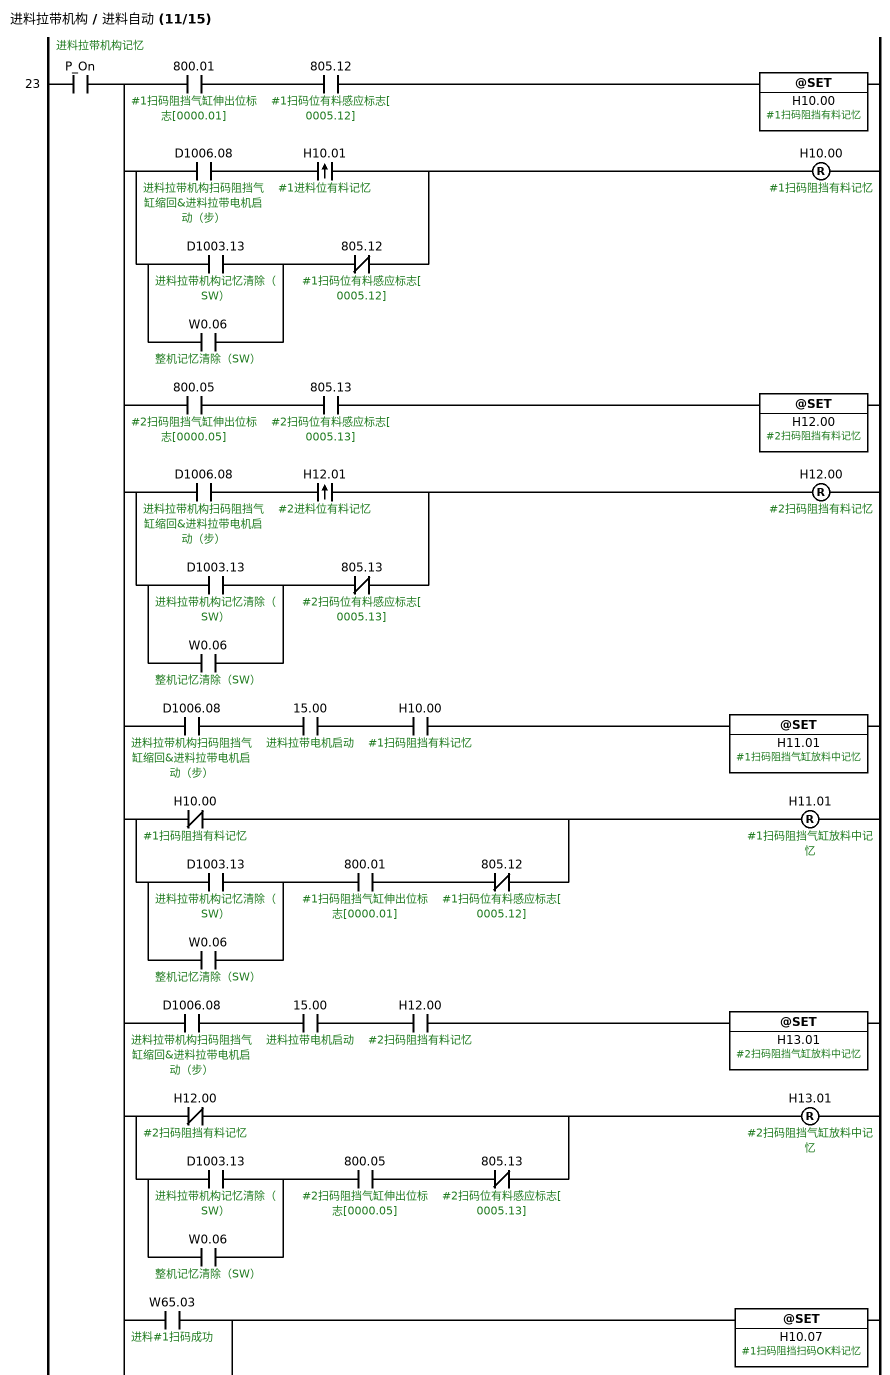
; [picture p48: 进料拉带机构 / 进料自动, rungs 23-23]

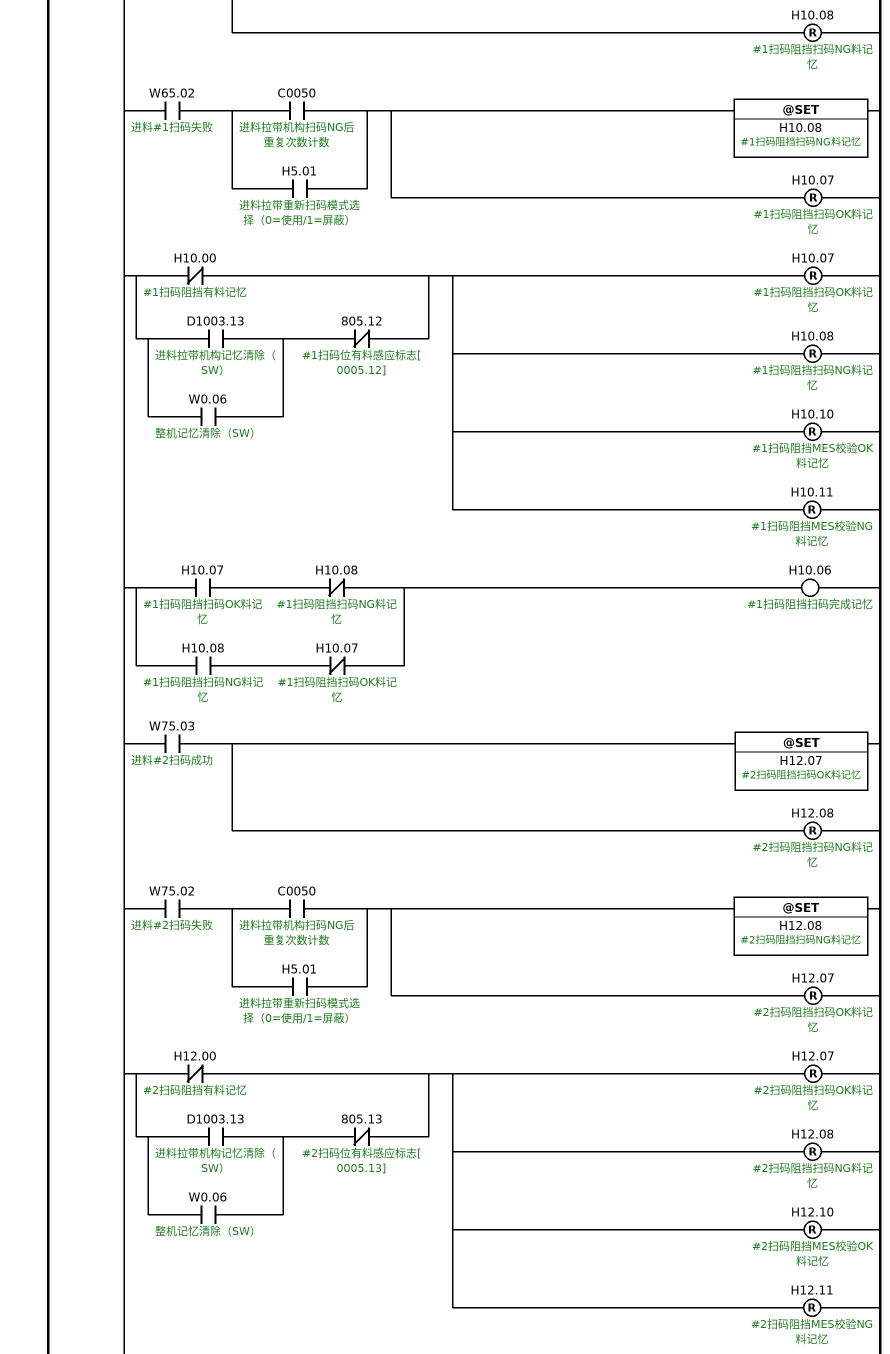

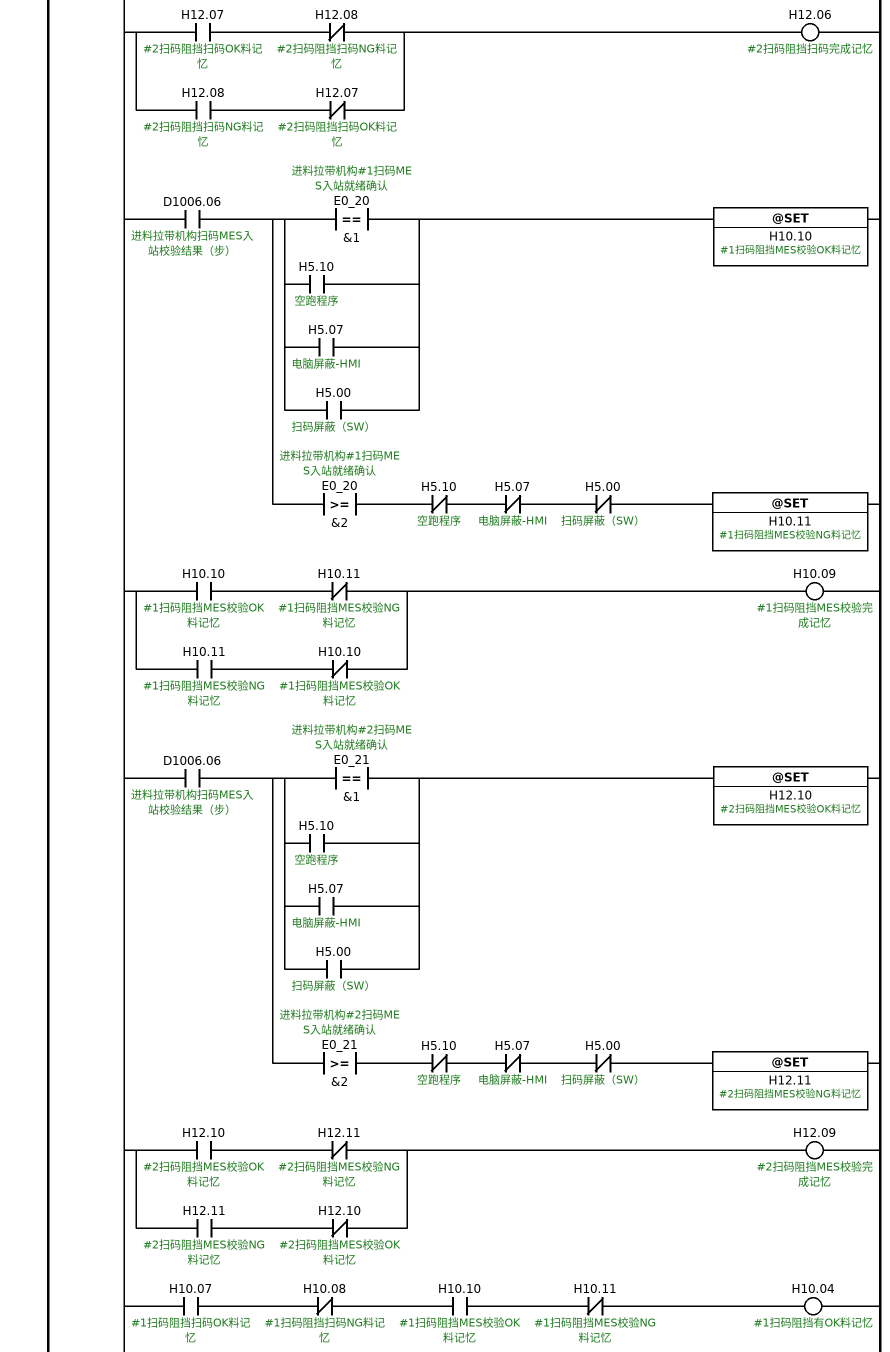

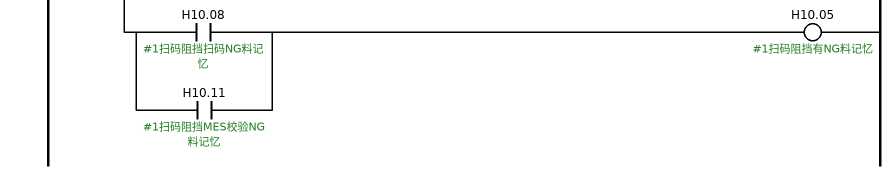
; rung 23: 进料拉带机构记忆
LD P_On
OUT TR0
AND 800.01  ; #1扫码阻挡气缸伸出位标志[0000.01]
AND 805.12  ; #1扫码位有料感应标志[0005.12]
@SET H10.00  ; #1扫码阻挡有料记忆
LD TR0
LD D1006.08  ; 进料拉带机构扫码阻挡气缸缩回&进料拉带电机启动（步）
@AND H10.01  ; #1进料位有料记忆
LD D1003.13  ; 进料拉带机构记忆清除（SW）
OR W0.06  ; 整机记忆清除（SW）
ANDNOT 805.12  ; #1扫码位有料感应标志[0005.12]
ORLD
ANDLD
RSET H10.00  ; #1扫码阻挡有料记忆
LD TR0
AND 800.05  ; #2扫码阻挡气缸伸出位标志[0000.05]
AND 805.13  ; #2扫码位有料感应标志[0005.13]
@SET H12.00  ; #2扫码阻挡有料记忆
LD TR0
LD D1006.08  ; 进料拉带机构扫码阻挡气缸缩回&进料拉带电机启动（步）
@AND H12.01  ; #2进料位有料记忆
LD D1003.13  ; 进料拉带机构记忆清除（SW）
OR W0.06  ; 整机记忆清除（SW）
ANDNOT 805.13  ; #2扫码位有料感应标志[0005.13]
ORLD
ANDLD
RSET H12.00  ; #2扫码阻挡有料记忆
LD TR0
AND D1006.08  ; 进料拉带机构扫码阻挡气缸缩回&进料拉带电机启动（步）
AND 15.00  ; 进料拉带电机启动
AND H10.00  ; #1扫码阻挡有料记忆
@SET H11.01  ; #1扫码阻挡气缸放料中记忆
LD TR0
LDNOT H10.00  ; #1扫码阻挡有料记忆
LD D1003.13  ; 进料拉带机构记忆清除（SW）
OR W0.06  ; 整机记忆清除（SW）
AND 800.01  ; #1扫码阻挡气缸伸出位标志[0000.01]
ANDNOT 805.12  ; #1扫码位有料感应标志[0005.12]
ORLD
ANDLD
RSET H11.01  ; #1扫码阻挡气缸放料中记忆
LD TR0
AND D1006.08  ; 进料拉带机构扫码阻挡气缸缩回&进料拉带电机启动（步）
AND 15.00  ; 进料拉带电机启动
AND H12.00  ; #2扫码阻挡有料记忆
@SET H13.01  ; #2扫码阻挡气缸放料中记忆
LD TR0
LDNOT H12.00  ; #2扫码阻挡有料记忆
LD D1003.13  ; 进料拉带机构记忆清除（SW）
OR W0.06  ; 整机记忆清除（SW）
AND 800.05  ; #2扫码阻挡气缸伸出位标志[0000.05]
ANDNOT 805.13  ; #2扫码位有料感应标志[0005.13]
ORLD
ANDLD
RSET H13.01  ; #2扫码阻挡气缸放料中记忆
LD TR0
AND W65.03  ; 进料#1扫码成功
@SET H10.07  ; #1扫码阻挡扫码OK料记忆
RSET H10.08  ; #1扫码阻挡扫码NG料记忆
LD TR0
AND W65.02  ; 进料#1扫码失败
LD C0050  ; 进料拉带机构扫码NG后重复次数计数
OR H5.01  ; 进料拉带重新扫码模式选择（0=使用/1=屏蔽）
ANDLD
@SET H10.08  ; #1扫码阻挡扫码NG料记忆
RSET H10.07  ; #1扫码阻挡扫码OK料记忆
LD TR0
LDNOT H10.00  ; #1扫码阻挡有料记忆
LD D1003.13  ; 进料拉带机构记忆清除（SW）
OR W0.06  ; 整机记忆清除（SW）
ANDNOT 805.12  ; #1扫码位有料感应标志[0005.12]
ORLD
ANDLD
RSET H10.07  ; #1扫码阻挡扫码OK料记忆
RSET H10.08  ; #1扫码阻挡扫码NG料记忆
RSET H10.10  ; #1扫码阻挡MES校验OK料记忆
RSET H10.11  ; #1扫码阻挡MES校验NG料记忆
LD TR0
LD H10.07  ; #1扫码阻挡扫码OK料记忆
ANDNOT H10.08  ; #1扫码阻挡扫码NG料记忆
LD H10.08  ; #1扫码阻挡扫码NG料记忆
ANDNOT H10.07  ; #1扫码阻挡扫码OK料记忆
ORLD
ANDLD
OUT H10.06  ; #1扫码阻挡扫码完成记忆
LD TR0
AND W75.03  ; 进料#2扫码成功
@SET H12.07  ; #2扫码阻挡扫码OK料记忆
RSET H12.08  ; #2扫码阻挡扫码NG料记忆
LD TR0
AND W75.02  ; 进料#2扫码失败
LD C0050  ; 进料拉带机构扫码NG后重复次数计数
OR H5.01  ; 进料拉带重新扫码模式选择（0=使用/1=屏蔽）
ANDLD
@SET H12.08  ; #2扫码阻挡扫码NG料记忆
RSET H12.07  ; #2扫码阻挡扫码OK料记忆
LD TR0
LDNOT H12.00  ; #2扫码阻挡有料记忆
LD D1003.13  ; 进料拉带机构记忆清除（SW）
OR W0.06  ; 整机记忆清除（SW）
ANDNOT 805.13  ; #2扫码位有料感应标志[0005.13]
ORLD
ANDLD
RSET H12.07  ; #2扫码阻挡扫码OK料记忆
RSET H12.08  ; #2扫码阻挡扫码NG料记忆
RSET H12.10  ; #2扫码阻挡MES校验OK料记忆
RSET H12.11  ; #2扫码阻挡MES校验NG料记忆
LD TR0
LD H12.07  ; #2扫码阻挡扫码OK料记忆
ANDNOT H12.08  ; #2扫码阻挡扫码NG料记忆
LD H12.08  ; #2扫码阻挡扫码NG料记忆
ANDNOT H12.07  ; #2扫码阻挡扫码OK料记忆
ORLD
ANDLD
OUT H12.06  ; #2扫码阻挡扫码完成记忆
LD TR0
AND D1006.06  ; 进料拉带机构扫码MES入站校验结果（步）
OUT TR1
LD=(300) E0_20 &1  ; 进料拉带机构#1扫码MES入站就绪确认  // 入站就绪确认=0：未确认，1：确认OK，2：确认NG
OR H5.10  ; 空跑程序
OR H5.07  ; 电脑屏蔽-HMI
OR H5.00  ; 扫码屏蔽（SW）
ANDLD
@SET H10.10  ; #1扫码阻挡MES校验OK料记忆
LD TR1
AND>=(325) E0_20 &2  ; 进料拉带机构#1扫码MES入站就绪确认  // 入站就绪确认=0：未确认，1：确认OK，2：确认NG
ANDNOT H5.10  ; 空跑程序
ANDNOT H5.07  ; 电脑屏蔽-HMI
ANDNOT H5.00  ; 扫码屏蔽（SW）
@SET H10.11  ; #1扫码阻挡MES校验NG料记忆
LD TR0
LD H10.10  ; #1扫码阻挡MES校验OK料记忆
ANDNOT H10.11  ; #1扫码阻挡MES校验NG料记忆
LD H10.11  ; #1扫码阻挡MES校验NG料记忆
ANDNOT H10.10  ; #1扫码阻挡MES校验OK料记忆
ORLD
ANDLD
OUT H10.09  ; #1扫码阻挡MES校验完成记忆
LD TR0
AND D1006.06  ; 进料拉带机构扫码MES入站校验结果（步）
OUT TR1
LD=(300) E0_21 &1  ; 进料拉带机构#2扫码MES入站就绪确认  // 入站就绪确认=0：未确认，1：确认OK，2：确认NG
OR H5.10  ; 空跑程序
OR H5.07  ; 电脑屏蔽-HMI
OR H5.00  ; 扫码屏蔽（SW）
ANDLD
@SET H12.10  ; #2扫码阻挡MES校验OK料记忆
LD TR1
AND>=(325) E0_21 &2  ; 进料拉带机构#2扫码MES入站就绪确认  // 入站就绪确认=0：未确认，1：确认OK，2：确认NG
ANDNOT H5.10  ; 空跑程序
ANDNOT H5.07  ; 电脑屏蔽-HMI
ANDNOT H5.00  ; 扫码屏蔽（SW）
@SET H12.11  ; #2扫码阻挡MES校验NG料记忆
LD TR0
LD H12.10  ; #2扫码阻挡MES校验OK料记忆
ANDNOT H12.11  ; #2扫码阻挡MES校验NG料记忆
LD H12.11  ; #2扫码阻挡MES校验NG料记忆
ANDNOT H12.10  ; #2扫码阻挡MES校验OK料记忆
ORLD
ANDLD
OUT H12.09  ; #2扫码阻挡MES校验完成记忆
LD TR0
AND H10.07  ; #1扫码阻挡扫码OK料记忆
ANDNOT H10.08  ; #1扫码阻挡扫码NG料记忆
AND H10.10  ; #1扫码阻挡MES校验OK料记忆
ANDNOT H10.11  ; #1扫码阻挡MES校验NG料记忆
OUT H10.04  ; #1扫码阻挡有OK料记忆
LD TR0
LD H10.08  ; #1扫码阻挡扫码NG料记忆
OR H10.11  ; #1扫码阻挡MES校验NG料记忆
ANDLD
OUT H10.05  ; #1扫码阻挡有NG料记忆

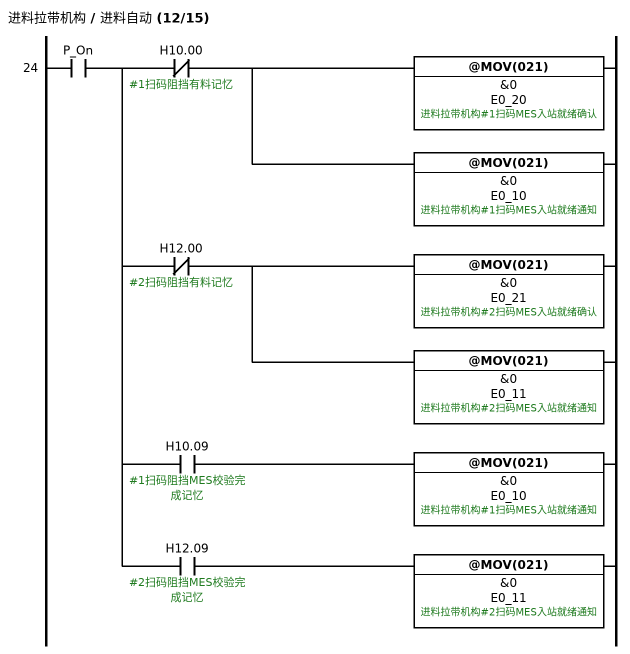
; rung 24
LD P_On
OUT TR0
ANDNOT H10.00  ; #1扫码阻挡有料记忆
@MOV(021) &0 E0_20  ; 进料拉带机构#1扫码MES入站就绪确认
@MOV(021) &0 E0_10  ; 进料拉带机构#1扫码MES入站就绪通知
LD TR0
ANDNOT H12.00  ; #2扫码阻挡有料记忆
@MOV(021) &0 E0_21  ; 进料拉带机构#2扫码MES入站就绪确认
@MOV(021) &0 E0_11  ; 进料拉带机构#2扫码MES入站就绪通知
LD TR0
AND H10.09  ; #1扫码阻挡MES校验完成记忆
@MOV(021) &0 E0_10  ; 进料拉带机构#1扫码MES入站就绪通知
LD TR0
AND H12.09  ; #2扫码阻挡MES校验完成记忆
@MOV(021) &0 E0_11  ; 进料拉带机构#2扫码MES入站就绪通知

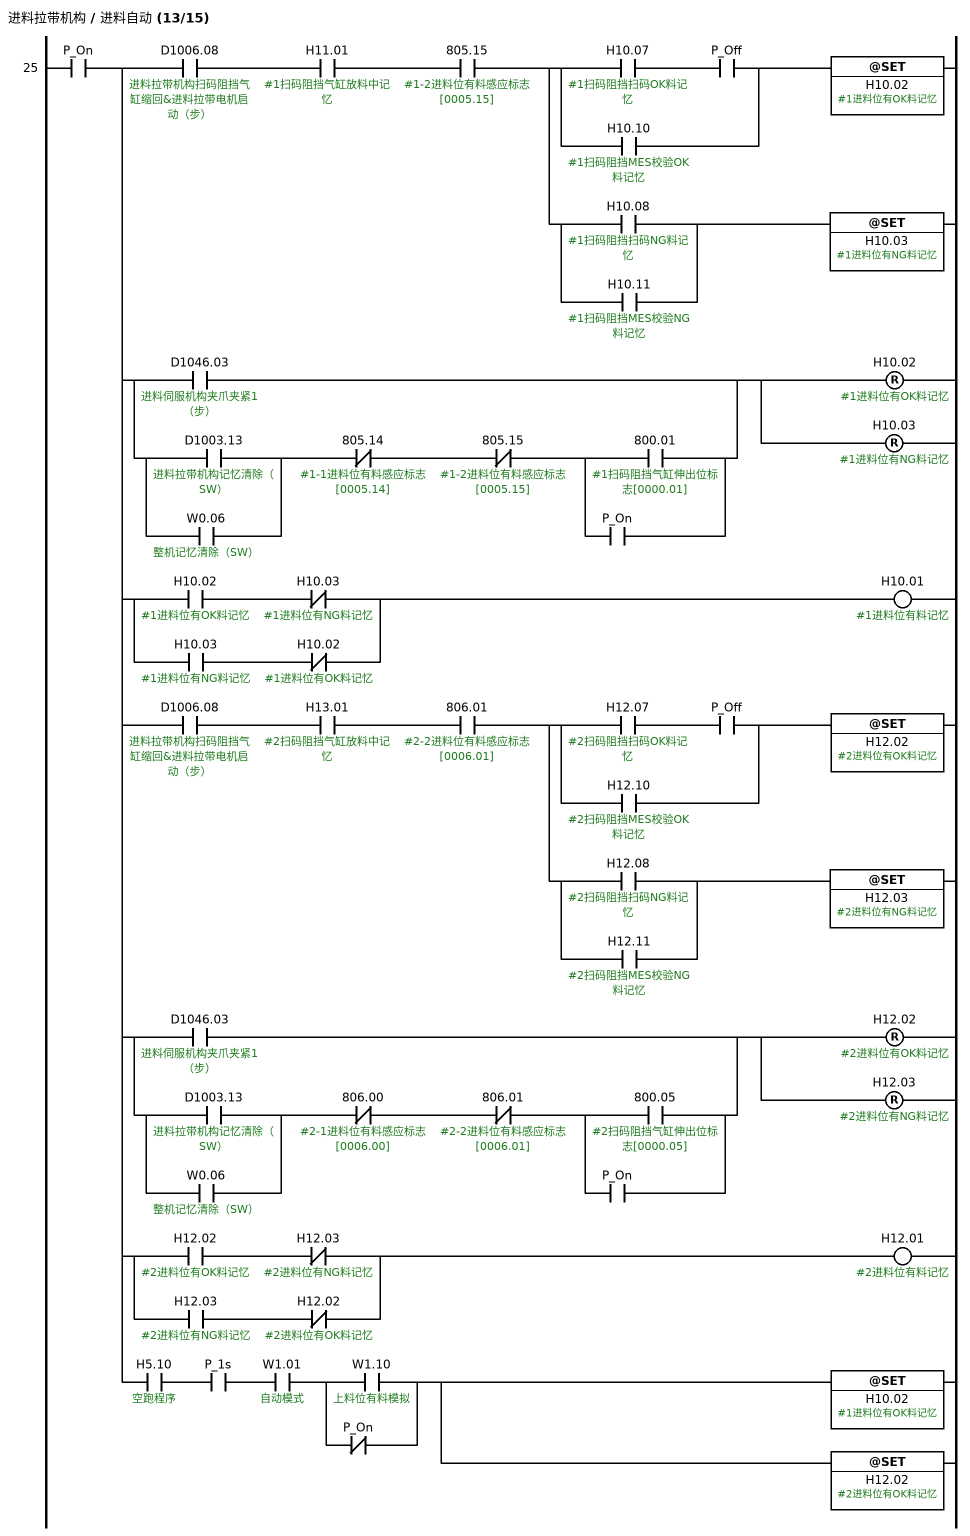
; rung 25
LD P_On
OUT TR0
AND D1006.08  ; 进料拉带机构扫码阻挡气缸缩回&进料拉带电机启动（步）
AND H11.01  ; #1扫码阻挡气缸放料中记忆
AND 805.15  ; #1-2进料位有料感应标志[0005.15]
OUT TR1
LD H10.07  ; #1扫码阻挡扫码OK料记忆
AND P_Off
OR H10.10  ; #1扫码阻挡MES校验OK料记忆
ANDLD
@SET H10.02  ; #1进料位有OK料记忆
LD TR1
LD H10.08  ; #1扫码阻挡扫码NG料记忆
OR H10.11  ; #1扫码阻挡MES校验NG料记忆
ANDLD
@SET H10.03  ; #1进料位有NG料记忆
LD TR0
LD D1046.03  ; 进料伺服机构夹爪夹紧1（步）
LD D1003.13  ; 进料拉带机构记忆清除（SW）
OR W0.06  ; 整机记忆清除（SW）
ANDNOT 805.14  ; #1-1进料位有料感应标志[0005.14]
ANDNOT 805.15  ; #1-2进料位有料感应标志[0005.15]
LD 800.01  ; #1扫码阻挡气缸伸出位标志[0000.01]
OR P_On
ANDLD
ORLD
ANDLD
RSET H10.02  ; #1进料位有OK料记忆
RSET H10.03  ; #1进料位有NG料记忆
LD TR0
LD H10.02  ; #1进料位有OK料记忆
ANDNOT H10.03  ; #1进料位有NG料记忆
LD H10.03  ; #1进料位有NG料记忆
ANDNOT H10.02  ; #1进料位有OK料记忆
ORLD
ANDLD
OUT H10.01  ; #1进料位有料记忆
LD TR0
AND D1006.08  ; 进料拉带机构扫码阻挡气缸缩回&进料拉带电机启动（步）
AND H13.01  ; #2扫码阻挡气缸放料中记忆
AND 806.01  ; #2-2进料位有料感应标志[0006.01]
OUT TR1
LD H12.07  ; #2扫码阻挡扫码OK料记忆
AND P_Off
OR H12.10  ; #2扫码阻挡MES校验OK料记忆
ANDLD
@SET H12.02  ; #2进料位有OK料记忆
LD TR1
LD H12.08  ; #2扫码阻挡扫码NG料记忆
OR H12.11  ; #2扫码阻挡MES校验NG料记忆
ANDLD
@SET H12.03  ; #2进料位有NG料记忆
LD TR0
LD D1046.03  ; 进料伺服机构夹爪夹紧1（步）
LD D1003.13  ; 进料拉带机构记忆清除（SW）
OR W0.06  ; 整机记忆清除（SW）
ANDNOT 806.00  ; #2-1进料位有料感应标志[0006.00]
ANDNOT 806.01  ; #2-2进料位有料感应标志[0006.01]
LD 800.05  ; #2扫码阻挡气缸伸出位标志[0000.05]
OR P_On
ANDLD
ORLD
ANDLD
RSET H12.02  ; #2进料位有OK料记忆
RSET H12.03  ; #2进料位有NG料记忆
LD TR0
LD H12.02  ; #2进料位有OK料记忆
ANDNOT H12.03  ; #2进料位有NG料记忆
LD H12.03  ; #2进料位有NG料记忆
ANDNOT H12.02  ; #2进料位有OK料记忆
ORLD
ANDLD
OUT H12.01  ; #2进料位有料记忆
LD TR0
AND H5.10  ; 空跑程序
AND P_1s
AND W1.01  ; 自动模式
LD W1.10  ; 上料位有料模拟
ORNOT P_On
ANDLD
@SET H10.02  ; #1进料位有OK料记忆
@SET H12.02  ; #2进料位有OK料记忆

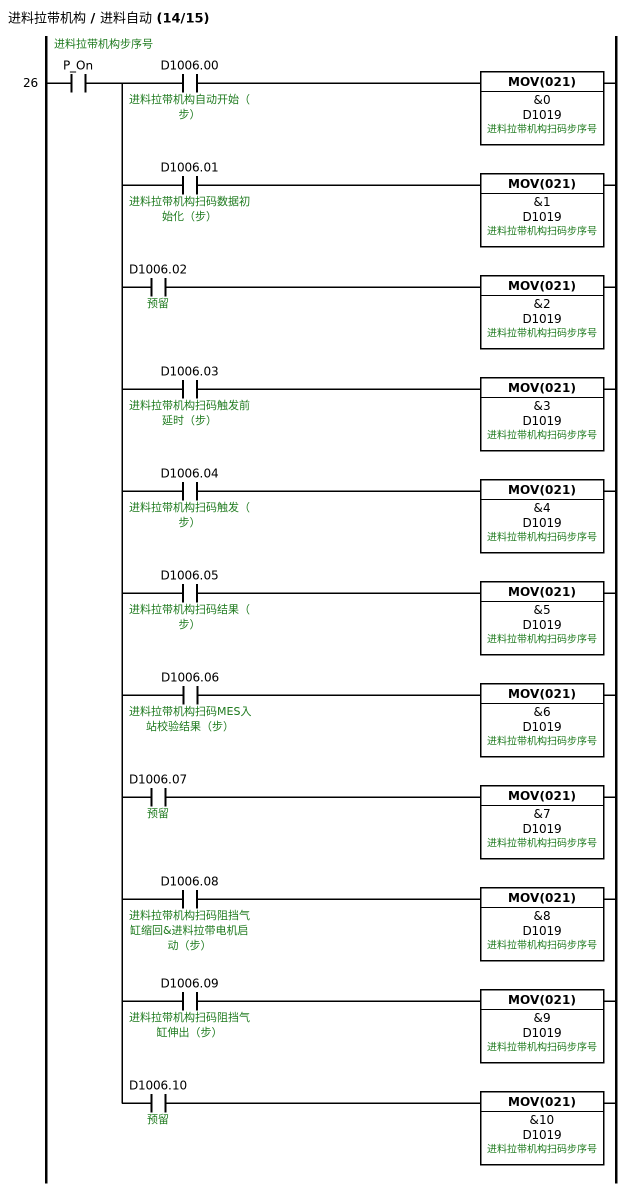
; rung 26: 进料拉带机构步序号
LD P_On
OUT TR0
AND D1006.00  ; 进料拉带机构自动开始（步）
MOV(021) &0 D1019  ; 进料拉带机构扫码步序号
LD TR0
AND D1006.01  ; 进料拉带机构扫码数据初始化（步）
MOV(021) &1 D1019  ; 进料拉带机构扫码步序号
LD TR0
AND D1006.02  ; 预留
MOV(021) &2 D1019  ; 进料拉带机构扫码步序号
LD TR0
AND D1006.03  ; 进料拉带机构扫码触发前延时（步）
MOV(021) &3 D1019  ; 进料拉带机构扫码步序号
LD TR0
AND D1006.04  ; 进料拉带机构扫码触发（步）
MOV(021) &4 D1019  ; 进料拉带机构扫码步序号
LD TR0
AND D1006.05  ; 进料拉带机构扫码结果（步）
MOV(021) &5 D1019  ; 进料拉带机构扫码步序号
LD TR0
AND D1006.06  ; 进料拉带机构扫码MES入站校验结果（步）
MOV(021) &6 D1019  ; 进料拉带机构扫码步序号
LD TR0
AND D1006.07  ; 预留
MOV(021) &7 D1019  ; 进料拉带机构扫码步序号
LD TR0
AND D1006.08  ; 进料拉带机构扫码阻挡气缸缩回&进料拉带电机启动（步）
MOV(021) &8 D1019  ; 进料拉带机构扫码步序号
LD TR0
AND D1006.09  ; 进料拉带机构扫码阻挡气缸伸出（步）
MOV(021) &9 D1019  ; 进料拉带机构扫码步序号
LD TR0
AND D1006.10  ; 预留
MOV(021) &10 D1019  ; 进料拉带机构扫码步序号

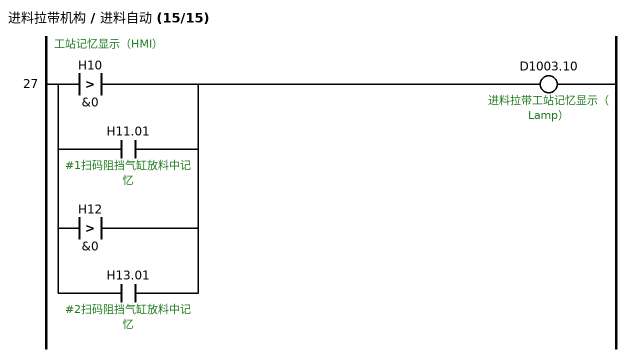
; rung 27: 工站记忆显示（HMI）
LD>(320) H10 &0
OR H11.01  ; #1扫码阻挡气缸放料中记忆
OR>(320) H12 &0
OR H13.01  ; #2扫码阻挡气缸放料中记忆
OUT D1003.10  ; 进料拉带工站记忆显示（Lamp）

### Section 工站复位

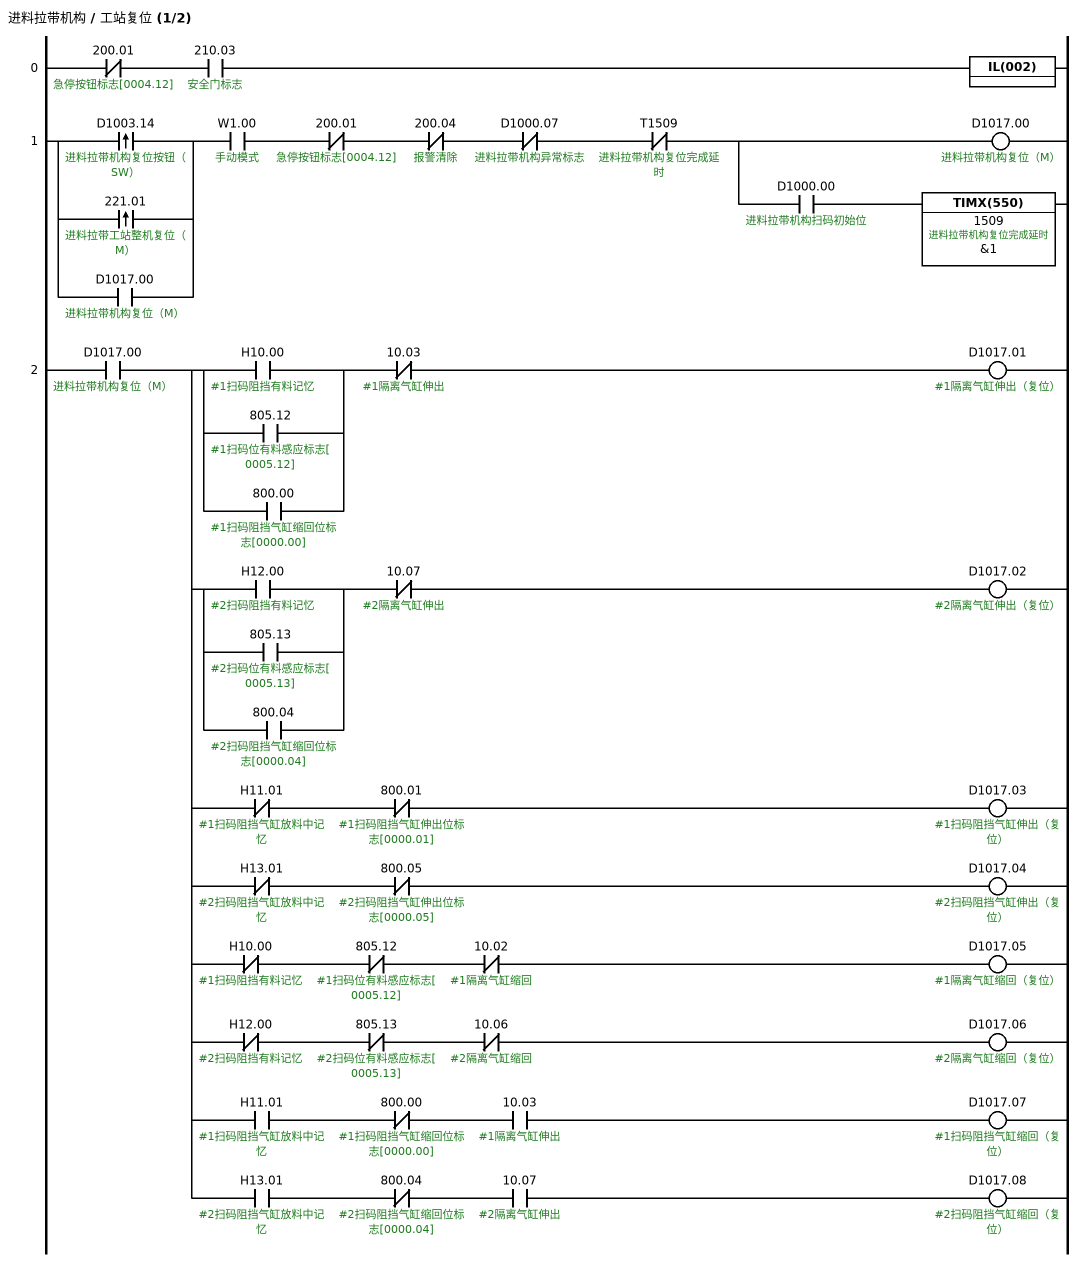
; rung 0
LDNOT 200.01  ; 急停按钮标志[0004.12]
AND 210.03  ; 安全门标志
IL(002)
; rung 1
@LD D1003.14  ; 进料拉带机构复位按钮（SW）
@OR 221.01  ; 进料拉带工站整机复位（M）
OR D1017.00  ; 进料拉带机构复位（M）
AND W1.00  ; 手动模式
ANDNOT 200.01  ; 急停按钮标志[0004.12]
ANDNOT 200.04  ; 报警清除
ANDNOT D1000.07  ; 进料拉带机构异常标志
ANDNOT T1509  ; 进料拉带机构复位完成延时
OUT D1017.00  ; 进料拉带机构复位（M）
AND D1000.00  ; 进料拉带机构扫码初始位
TIMX(550) 1509 &1  ; 进料拉带机构复位完成延时
; rung 2
LD D1017.00  ; 进料拉带机构复位（M）
OUT TR0
LD H10.00  ; #1扫码阻挡有料记忆
OR 805.12  ; #1扫码位有料感应标志[0005.12]
OR 800.00  ; #1扫码阻挡气缸缩回位标志[0000.00]
ANDLD
ANDNOT 10.03  ; #1隔离气缸伸出
OUT D1017.01  ; #1隔离气缸伸出（复位）
LD TR0
LD H12.00  ; #2扫码阻挡有料记忆
OR 805.13  ; #2扫码位有料感应标志[0005.13]
OR 800.04  ; #2扫码阻挡气缸缩回位标志[0000.04]
ANDLD
ANDNOT 10.07  ; #2隔离气缸伸出
OUT D1017.02  ; #2隔离气缸伸出（复位）
LD TR0
ANDNOT H11.01  ; #1扫码阻挡气缸放料中记忆
ANDNOT 800.01  ; #1扫码阻挡气缸伸出位标志[0000.01]
OUT D1017.03  ; #1扫码阻挡气缸伸出（复位）
LD TR0
ANDNOT H13.01  ; #2扫码阻挡气缸放料中记忆
ANDNOT 800.05  ; #2扫码阻挡气缸伸出位标志[0000.05]
OUT D1017.04  ; #2扫码阻挡气缸伸出（复位）
LD TR0
ANDNOT H10.00  ; #1扫码阻挡有料记忆
ANDNOT 805.12  ; #1扫码位有料感应标志[0005.12]
ANDNOT 10.02  ; #1隔离气缸缩回
OUT D1017.05  ; #1隔离气缸缩回（复位）
LD TR0
ANDNOT H12.00  ; #2扫码阻挡有料记忆
ANDNOT 805.13  ; #2扫码位有料感应标志[0005.13]
ANDNOT 10.06  ; #2隔离气缸缩回
OUT D1017.06  ; #2隔离气缸缩回（复位）
LD TR0
AND H11.01  ; #1扫码阻挡气缸放料中记忆
ANDNOT 800.00  ; #1扫码阻挡气缸缩回位标志[0000.00]
AND 10.03  ; #1隔离气缸伸出
OUT D1017.07  ; #1扫码阻挡气缸缩回（复位）
LD TR0
AND H13.01  ; #2扫码阻挡气缸放料中记忆
ANDNOT 800.04  ; #2扫码阻挡气缸缩回位标志[0000.04]
AND 10.07  ; #2隔离气缸伸出
OUT D1017.08  ; #2扫码阻挡气缸缩回（复位）

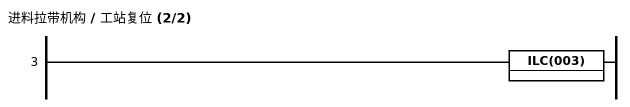
; rung 3
ILC(003)

### Section 指示灯

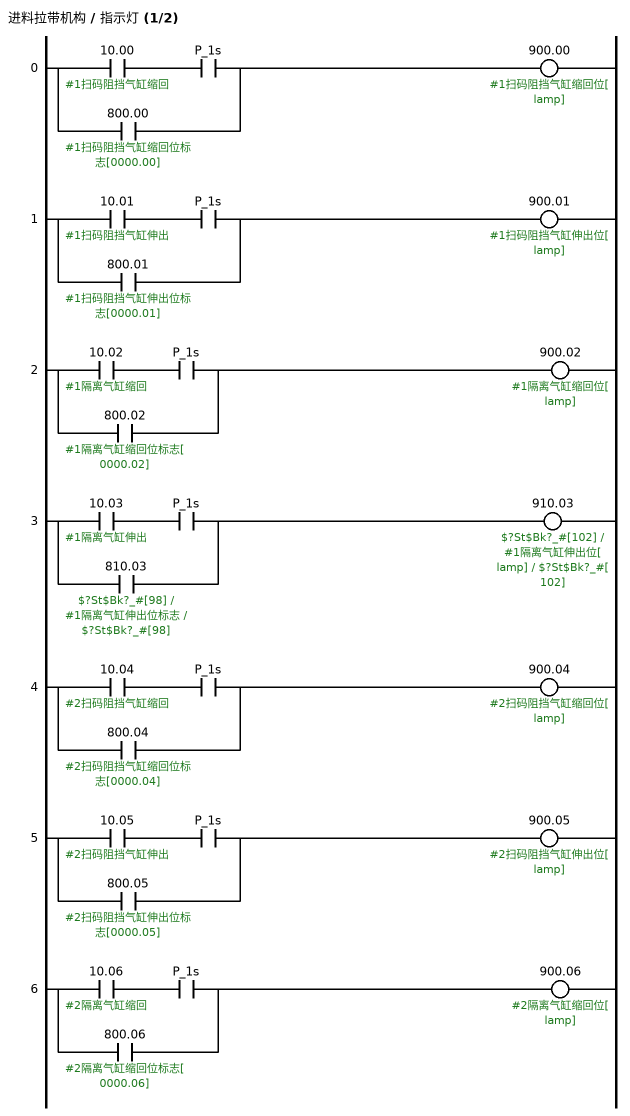
; rung 0
LD 10.00  ; #1扫码阻挡气缸缩回
AND P_1s
OR 800.00  ; #1扫码阻挡气缸缩回位标志[0000.00]
OUT 900.00  ; #1扫码阻挡气缸缩回位[lamp]
; rung 1
LD 10.01  ; #1扫码阻挡气缸伸出
AND P_1s
OR 800.01  ; #1扫码阻挡气缸伸出位标志[0000.01]
OUT 900.01  ; #1扫码阻挡气缸伸出位[lamp]
; rung 2
LD 10.02  ; #1隔离气缸缩回
AND P_1s
OR 800.02  ; #1隔离气缸缩回位标志[0000.02]
OUT 900.02  ; #1隔离气缸缩回位[lamp]
; rung 3
LD 10.03  ; #1隔离气缸伸出
AND P_1s
OR 810.03  ; $?St$Bk?_#[98] / #1隔离气缸伸出位标志 / $?St$Bk?_#[98]
OUT 910.03  ; $?St$Bk?_#[102] / #1隔离气缸伸出位[lamp] / $?St$Bk?_#[102]
; rung 4
LD 10.04  ; #2扫码阻挡气缸缩回
AND P_1s
OR 800.04  ; #2扫码阻挡气缸缩回位标志[0000.04]
OUT 900.04  ; #2扫码阻挡气缸缩回位[lamp]
; rung 5
LD 10.05  ; #2扫码阻挡气缸伸出
AND P_1s
OR 800.05  ; #2扫码阻挡气缸伸出位标志[0000.05]
OUT 900.05  ; #2扫码阻挡气缸伸出位[lamp]
; rung 6
LD 10.06  ; #2隔离气缸缩回
AND P_1s
OR 800.06  ; #2隔离气缸缩回位标志[0000.06]
OUT 900.06  ; #2隔离气缸缩回位[lamp]

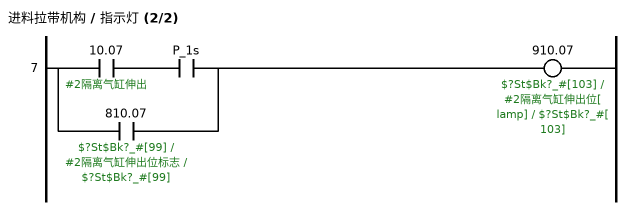
; rung 7
LD 10.07  ; #2隔离气缸伸出
AND P_1s
OR 810.07  ; $?St$Bk?_#[99] / #2隔离气缸伸出位标志 / $?St$Bk?_#[99]
OUT 910.07  ; $?St$Bk?_#[103] / #2隔离气缸伸出位[lamp] / $?St$Bk?_#[103]

### Section 外部输出

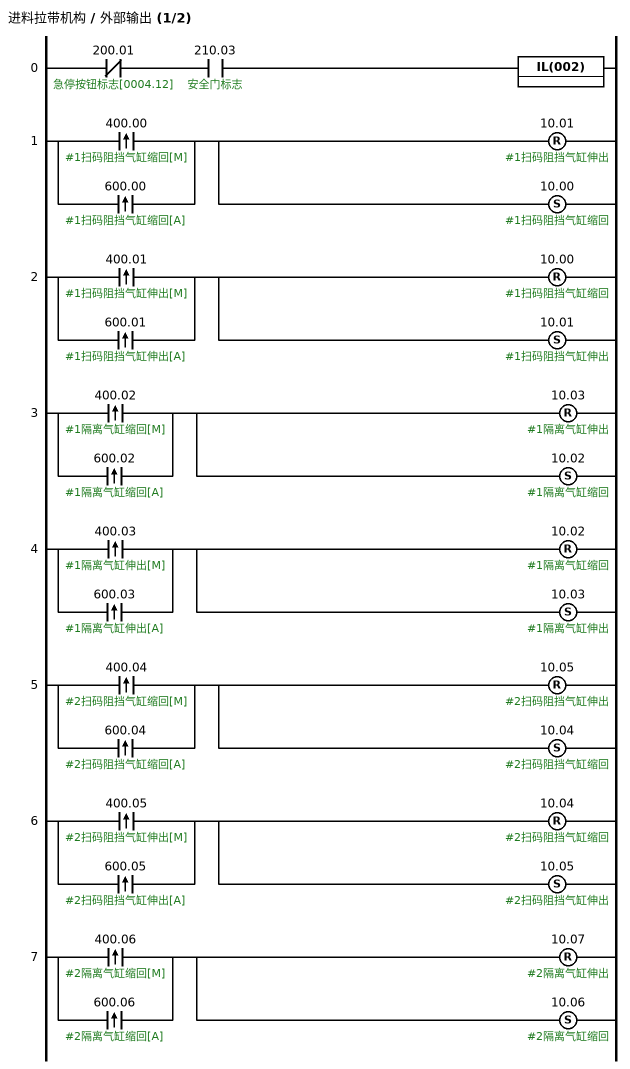
; rung 0
LDNOT 200.01  ; 急停按钮标志[0004.12]
AND 210.03  ; 安全门标志
IL(002)
; rung 1
@LD 400.00  ; #1扫码阻挡气缸缩回[M]
@OR 600.00  ; #1扫码阻挡气缸缩回[A]
RSET 10.01  ; #1扫码阻挡气缸伸出
SET 10.00  ; #1扫码阻挡气缸缩回
; rung 2
@LD 400.01  ; #1扫码阻挡气缸伸出[M]
@OR 600.01  ; #1扫码阻挡气缸伸出[A]
RSET 10.00  ; #1扫码阻挡气缸缩回
SET 10.01  ; #1扫码阻挡气缸伸出
; rung 3
@LD 400.02  ; #1隔离气缸缩回[M]
@OR 600.02  ; #1隔离气缸缩回[A]
RSET 10.03  ; #1隔离气缸伸出
SET 10.02  ; #1隔离气缸缩回
; rung 4
@LD 400.03  ; #1隔离气缸伸出[M]
@OR 600.03  ; #1隔离气缸伸出[A]
RSET 10.02  ; #1隔离气缸缩回
SET 10.03  ; #1隔离气缸伸出
; rung 5
@LD 400.04  ; #2扫码阻挡气缸缩回[M]
@OR 600.04  ; #2扫码阻挡气缸缩回[A]
RSET 10.05  ; #2扫码阻挡气缸伸出
SET 10.04  ; #2扫码阻挡气缸缩回
; rung 6
@LD 400.05  ; #2扫码阻挡气缸伸出[M]
@OR 600.05  ; #2扫码阻挡气缸伸出[A]
RSET 10.04  ; #2扫码阻挡气缸缩回
SET 10.05  ; #2扫码阻挡气缸伸出
; rung 7
@LD 400.06  ; #2隔离气缸缩回[M]
@OR 600.06  ; #2隔离气缸缩回[A]
RSET 10.07  ; #2隔离气缸伸出
SET 10.06  ; #2隔离气缸缩回

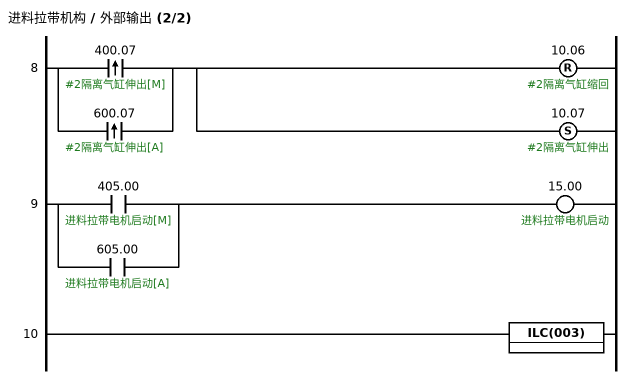
; rung 8
@LD 400.07  ; #2隔离气缸伸出[M]
@OR 600.07  ; #2隔离气缸伸出[A]
RSET 10.06  ; #2隔离气缸缩回
SET 10.07  ; #2隔离气缸伸出
; rung 9
LD 405.00  ; 进料拉带电机启动[M]
OR 605.00  ; 进料拉带电机启动[A]
OUT 15.00  ; 进料拉带电机启动
; rung 10
ILC(003)

### Section END
; rung 0
END(001)

## Program 进料伺服机构 (cyclic task 2)

### Section Main

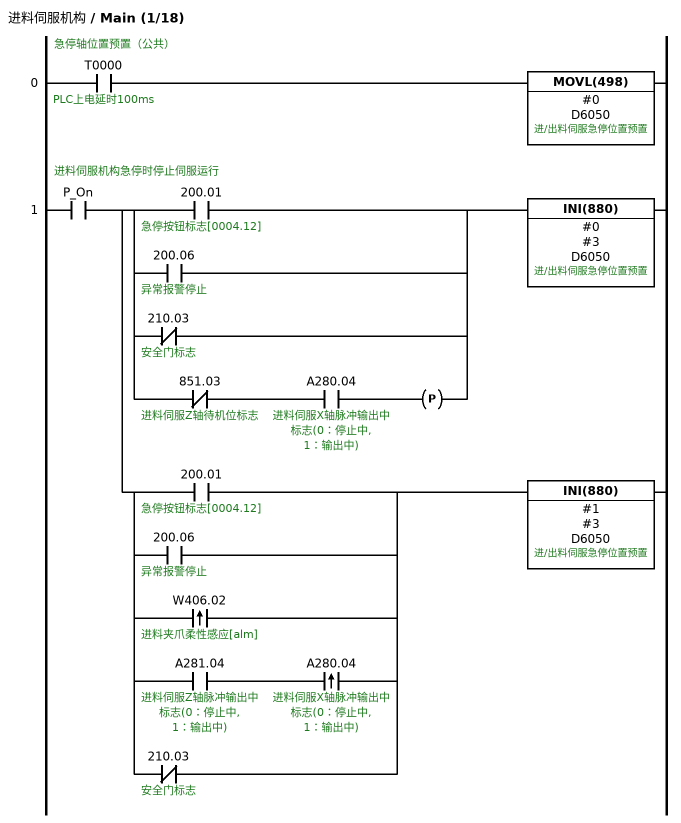
; rung 0: 急停轴位置预置（公共）
LD T0000  ; PLC上电延时100ms
MOVL(498) #0 D6050  ; 进/出料伺服急停位置预置
; rung 1: 进料伺服机构急停时停止伺服运行
LD P_On
OUT TR0
LD 200.01  ; 急停按钮标志[0004.12]
LD 200.06  ; 异常报警停止
ORNOT 210.03  ; 安全门标志
ORLD
LDNOT 851.03  ; 进料伺服Z轴待机位标志
AND A280.04  ; 进料伺服X轴脉冲输出中标志(0：停止中,1：输出中)
UP(521)
ORLD
ANDLD
INI(880) #0 #3 D6050  ; 进/出料伺服急停位置预置  // 进料X轴
LD TR0
LD 200.01  ; 急停按钮标志[0004.12]
OR 200.06  ; 异常报警停止
@OR W406.02  ; 进料夹爪柔性感应[alm]
LD A281.04  ; 进料伺服Z轴脉冲输出中标志(0：停止中,1：输出中)
@AND A280.04  ; 进料伺服X轴脉冲输出中标志(0：停止中,1：输出中)
ORLD
ORNOT 210.03  ; 安全门标志
ANDLD
INI(880) #1 #3 D6050  ; 进/出料伺服急停位置预置  // 进料Z轴

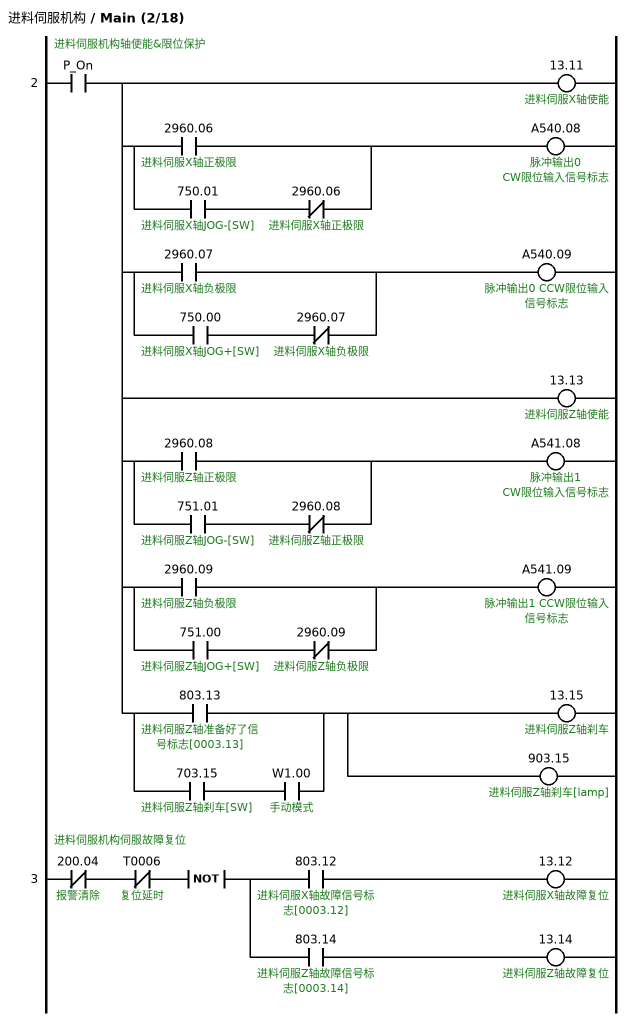
; rung 2: 进料伺服机构轴使能&限位保护
LD P_On
OUT TR0
OUT 13.11  ; 进料伺服X轴使能
LD 2960.06  ; 进料伺服X轴正极限
LD 750.01  ; 进料伺服X轴JOG-[SW]
ANDNOT 2960.06  ; 进料伺服X轴正极限
ORLD
ANDLD
OUT A540.08  ; 脉冲输出0 CW限位输入信号标志
LD TR0
LD 2960.07  ; 进料伺服X轴负极限
LD 750.00  ; 进料伺服X轴JOG+[SW]
ANDNOT 2960.07  ; 进料伺服X轴负极限
ORLD
ANDLD
OUT A540.09  ; 脉冲输出0 CCW限位输入信号标志
LD TR0
OUT 13.13  ; 进料伺服Z轴使能
LD 2960.08  ; 进料伺服Z轴正极限
LD 751.01  ; 进料伺服Z轴JOG-[SW]
ANDNOT 2960.08  ; 进料伺服Z轴正极限
ORLD
ANDLD
OUT A541.08  ; 脉冲输出1 CW限位输入信号标志
LD TR0
LD 2960.09  ; 进料伺服Z轴负极限
LD 751.00  ; 进料伺服Z轴JOG+[SW]
ANDNOT 2960.09  ; 进料伺服Z轴负极限
ORLD
ANDLD
OUT A541.09  ; 脉冲输出1 CCW限位输入信号标志
LD TR0
LD 803.13  ; 进料伺服Z轴准备好了信号标志[0003.13]
LD 703.15  ; 进料伺服Z轴刹车[SW]
AND W1.00  ; 手动模式
ORLD
ANDLD
OUT 13.15  ; 进料伺服Z轴刹车
OUT 903.15  ; 进料伺服Z轴刹车[lamp]
; rung 3: 进料伺服机构伺服故障复位
LDNOT 200.04  ; 报警清除
ANDNOT T0006  ; 复位延时
NOT(520)
OUT TR0
AND 803.12  ; 进料伺服X轴故障信号标志[0003.12]
OUT 13.12  ; 进料伺服X轴故障复位
LD TR0
AND 803.14  ; 进料伺服Z轴故障信号标志[0003.14]
OUT 13.14  ; 进料伺服Z轴故障复位

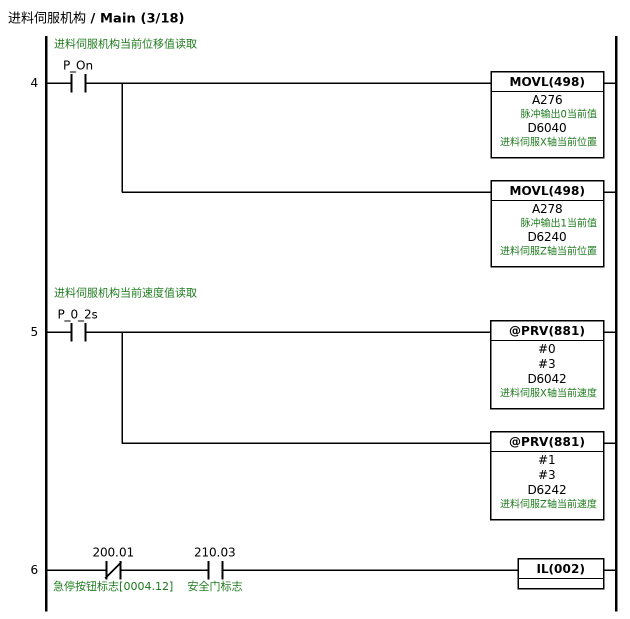
; rung 4: 进料伺服机构当前位移值读取
LD P_On
MOVL(498) A276 D6040  ; 脉冲输出0当前值, 进料伺服X轴当前位置
MOVL(498) A278 D6240  ; 脉冲输出1当前值, 进料伺服Z轴当前位置
; rung 5: 进料伺服机构当前速度值读取
LD P_0_2s
@PRV(881) #0 #3 D6042  ; 进料伺服X轴当前速度
@PRV(881) #1 #3 D6242  ; 进料伺服Z轴当前速度
; rung 6
LDNOT 200.01  ; 急停按钮标志[0004.12]
AND 210.03  ; 安全门标志
IL(002)

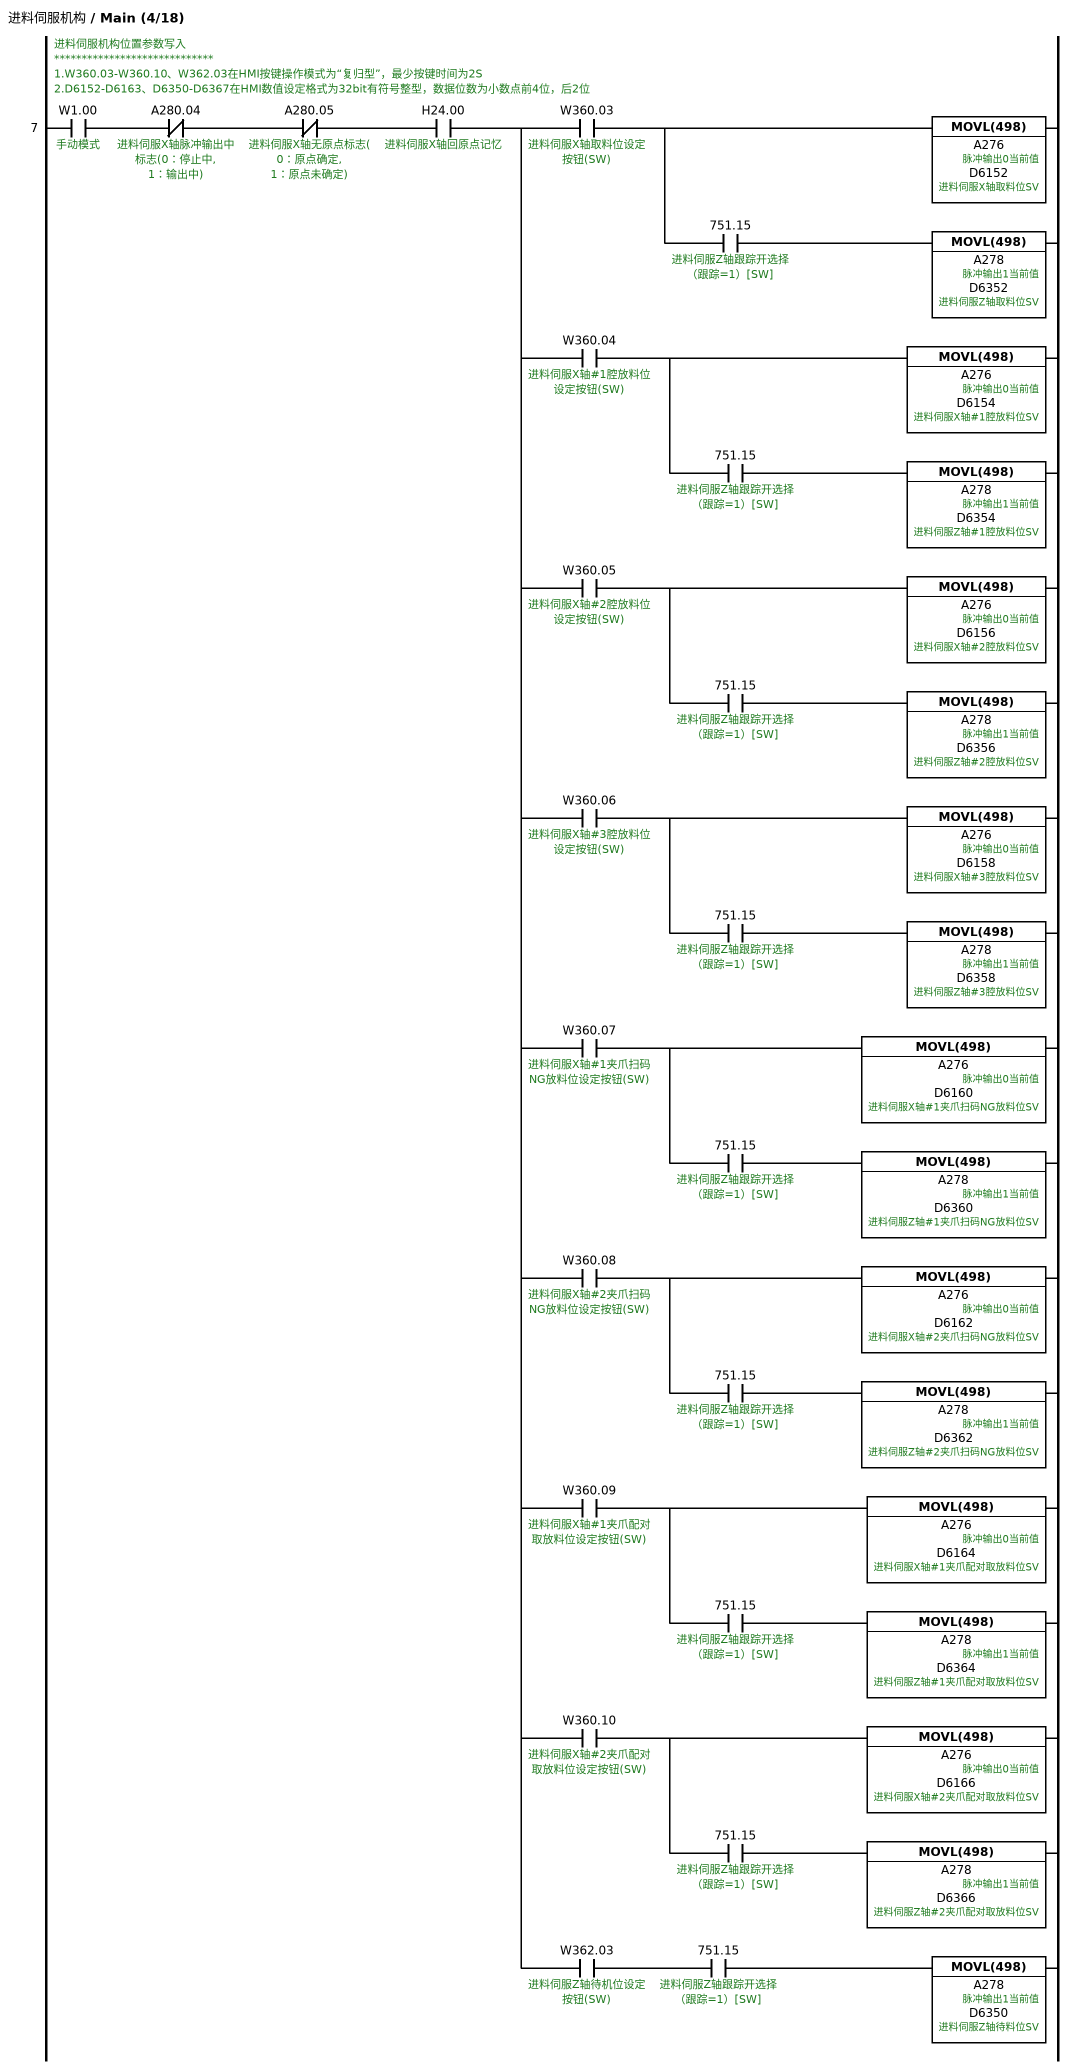
; rung 7: 进料伺服机构位置参数写入 / ***************************** / 1.W360.03-W360.10、W362.03在HMI按键操作模式为“复归型”，最少按键时间为2S / 2.D6152-D6163、D6350-D6367在HMI数值设定格式为32bit有符号整型，数据位数为小数点前4位，后2位
LD W1.00  ; 手动模式
ANDNOT A280.04  ; 进料伺服X轴脉冲输出中标志(0：停止中,1：输出中)
ANDNOT A280.05  ; 进料伺服X轴无原点标志(0：原点确定,1：原点未确定)
AND H24.00  ; 进料伺服X轴回原点记忆
OUT TR0
AND W360.03  ; 进料伺服X轴取料位设定按钮(SW)
MOVL(498) A276 D6152  ; 脉冲输出0当前值, 进料伺服X轴取料位SV
AND 751.15  ; 进料伺服Z轴跟踪开选择（跟踪=1）[SW]
MOVL(498) A278 D6352  ; 脉冲输出1当前值, 进料伺服Z轴取料位SV
LD TR0
AND W360.04  ; 进料伺服X轴#1腔放料位设定按钮(SW)
MOVL(498) A276 D6154  ; 脉冲输出0当前值, 进料伺服X轴#1腔放料位SV
AND 751.15  ; 进料伺服Z轴跟踪开选择（跟踪=1）[SW]
MOVL(498) A278 D6354  ; 脉冲输出1当前值, 进料伺服Z轴#1腔放料位SV
LD TR0
AND W360.05  ; 进料伺服X轴#2腔放料位设定按钮(SW)
MOVL(498) A276 D6156  ; 脉冲输出0当前值, 进料伺服X轴#2腔放料位SV
AND 751.15  ; 进料伺服Z轴跟踪开选择（跟踪=1）[SW]
MOVL(498) A278 D6356  ; 脉冲输出1当前值, 进料伺服Z轴#2腔放料位SV
LD TR0
AND W360.06  ; 进料伺服X轴#3腔放料位设定按钮(SW)
MOVL(498) A276 D6158  ; 脉冲输出0当前值, 进料伺服X轴#3腔放料位SV
AND 751.15  ; 进料伺服Z轴跟踪开选择（跟踪=1）[SW]
MOVL(498) A278 D6358  ; 脉冲输出1当前值, 进料伺服Z轴#3腔放料位SV
LD TR0
AND W360.07  ; 进料伺服X轴#1夹爪扫码NG放料位设定按钮(SW)
MOVL(498) A276 D6160  ; 脉冲输出0当前值, 进料伺服X轴#1夹爪扫码NG放料位SV
AND 751.15  ; 进料伺服Z轴跟踪开选择（跟踪=1）[SW]
MOVL(498) A278 D6360  ; 脉冲输出1当前值, 进料伺服Z轴#1夹爪扫码NG放料位SV
LD TR0
AND W360.08  ; 进料伺服X轴#2夹爪扫码NG放料位设定按钮(SW)
MOVL(498) A276 D6162  ; 脉冲输出0当前值, 进料伺服X轴#2夹爪扫码NG放料位SV
AND 751.15  ; 进料伺服Z轴跟踪开选择（跟踪=1）[SW]
MOVL(498) A278 D6362  ; 脉冲输出1当前值, 进料伺服Z轴#2夹爪扫码NG放料位SV
LD TR0
AND W360.09  ; 进料伺服X轴#1夹爪配对取放料位设定按钮(SW)
MOVL(498) A276 D6164  ; 脉冲输出0当前值, 进料伺服X轴#1夹爪配对取放料位SV
AND 751.15  ; 进料伺服Z轴跟踪开选择（跟踪=1）[SW]
MOVL(498) A278 D6364  ; 脉冲输出1当前值, 进料伺服Z轴#1夹爪配对取放料位SV
LD TR0
AND W360.10  ; 进料伺服X轴#2夹爪配对取放料位设定按钮(SW)
MOVL(498) A276 D6166  ; 脉冲输出0当前值, 进料伺服X轴#2夹爪配对取放料位SV
AND 751.15  ; 进料伺服Z轴跟踪开选择（跟踪=1）[SW]
MOVL(498) A278 D6366  ; 脉冲输出1当前值, 进料伺服Z轴#2夹爪配对取放料位SV
LD TR0
AND W362.03  ; 进料伺服Z轴待机位设定按钮(SW)
AND 751.15  ; 进料伺服Z轴跟踪开选择（跟踪=1）[SW]
MOVL(498) A278 D6350  ; 脉冲输出1当前值, 进料伺服Z轴待料位SV

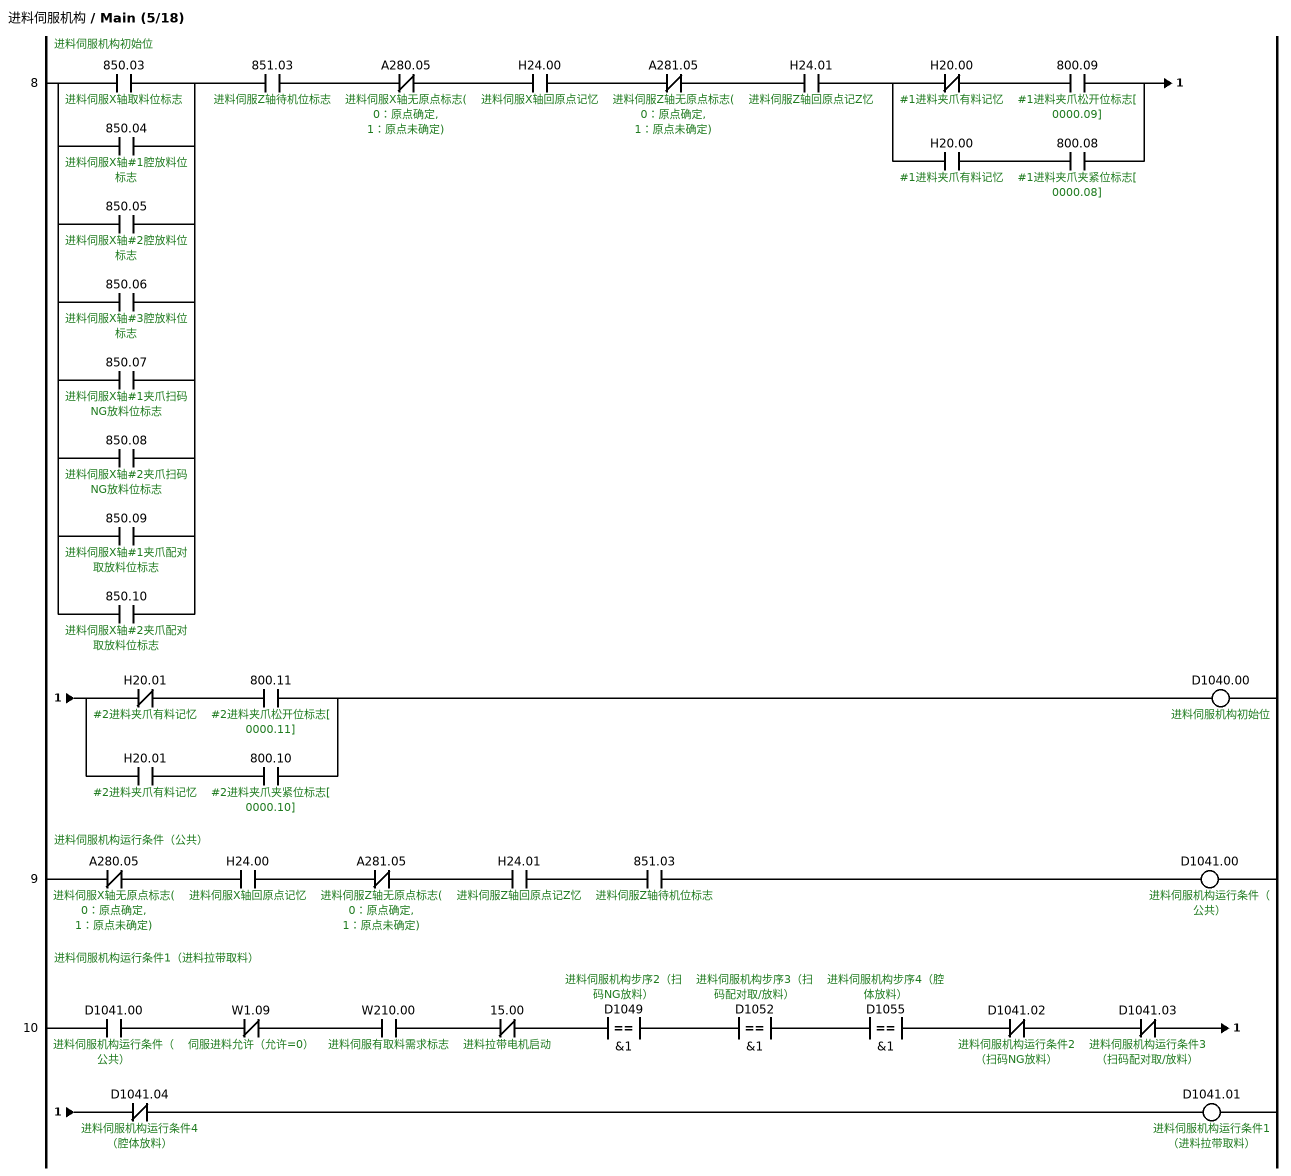
; rung 8: 进料伺服机构初始位
LD 850.03  ; 进料伺服X轴取料位标志
OR 850.04  ; 进料伺服X轴#1腔放料位标志
OR 850.05  ; 进料伺服X轴#2腔放料位标志
OR 850.06  ; 进料伺服X轴#3腔放料位标志
OR 850.07  ; 进料伺服X轴#1夹爪扫码NG放料位标志
OR 850.08  ; 进料伺服X轴#2夹爪扫码NG放料位标志
OR 850.09  ; 进料伺服X轴#1夹爪配对取放料位标志
OR 850.10  ; 进料伺服X轴#2夹爪配对取放料位标志
AND 851.03  ; 进料伺服Z轴待机位标志
ANDNOT A280.05  ; 进料伺服X轴无原点标志(0：原点确定,1：原点未确定)
AND H24.00  ; 进料伺服X轴回原点记忆
ANDNOT A281.05  ; 进料伺服Z轴无原点标志(0：原点确定,1：原点未确定)
AND H24.01  ; 进料伺服Z轴回原点记Z忆
LDNOT H20.00  ; #1进料夹爪有料记忆
AND 800.09  ; #1进料夹爪松开位标志[0000.09]
LD H20.00  ; #1进料夹爪有料记忆
AND 800.08  ; #1进料夹爪夹紧位标志[0000.08]
ORLD
ANDLD
LDNOT H20.01  ; #2进料夹爪有料记忆
AND 800.11  ; #2进料夹爪松开位标志[0000.11]
LD H20.01  ; #2进料夹爪有料记忆
AND 800.10  ; #2进料夹爪夹紧位标志[0000.10]
ORLD
ANDLD
OUT D1040.00  ; 进料伺服机构初始位
; rung 9: 进料伺服机构运行条件（公共）
LDNOT A280.05  ; 进料伺服X轴无原点标志(0：原点确定,1：原点未确定)
AND H24.00  ; 进料伺服X轴回原点记忆
ANDNOT A281.05  ; 进料伺服Z轴无原点标志(0：原点确定,1：原点未确定)
AND H24.01  ; 进料伺服Z轴回原点记Z忆
AND 851.03  ; 进料伺服Z轴待机位标志
OUT D1041.00  ; 进料伺服机构运行条件（公共）
; rung 10: 进料伺服机构运行条件1（进料拉带取料）
LD D1041.00  ; 进料伺服机构运行条件（公共）
ANDNOT W1.09  ; 伺服进料允许（允许=0）
AND W210.00  ; 进料伺服有取料需求标志
ANDNOT 15.00  ; 进料拉带电机启动
AND=(300) D1049 &1  ; 进料伺服机构步序2（扫码NG放料）
AND=(300) D1052 &1  ; 进料伺服机构步序3（扫码配对取/放料）
AND=(300) D1055 &1  ; 进料伺服机构步序4（腔体放料）
ANDNOT D1041.02  ; 进料伺服机构运行条件2（扫码NG放料）
ANDNOT D1041.03  ; 进料伺服机构运行条件3（扫码配对取/放料）
ANDNOT D1041.04  ; 进料伺服机构运行条件4（腔体放料）
OUT D1041.01  ; 进料伺服机构运行条件1（进料拉带取料）

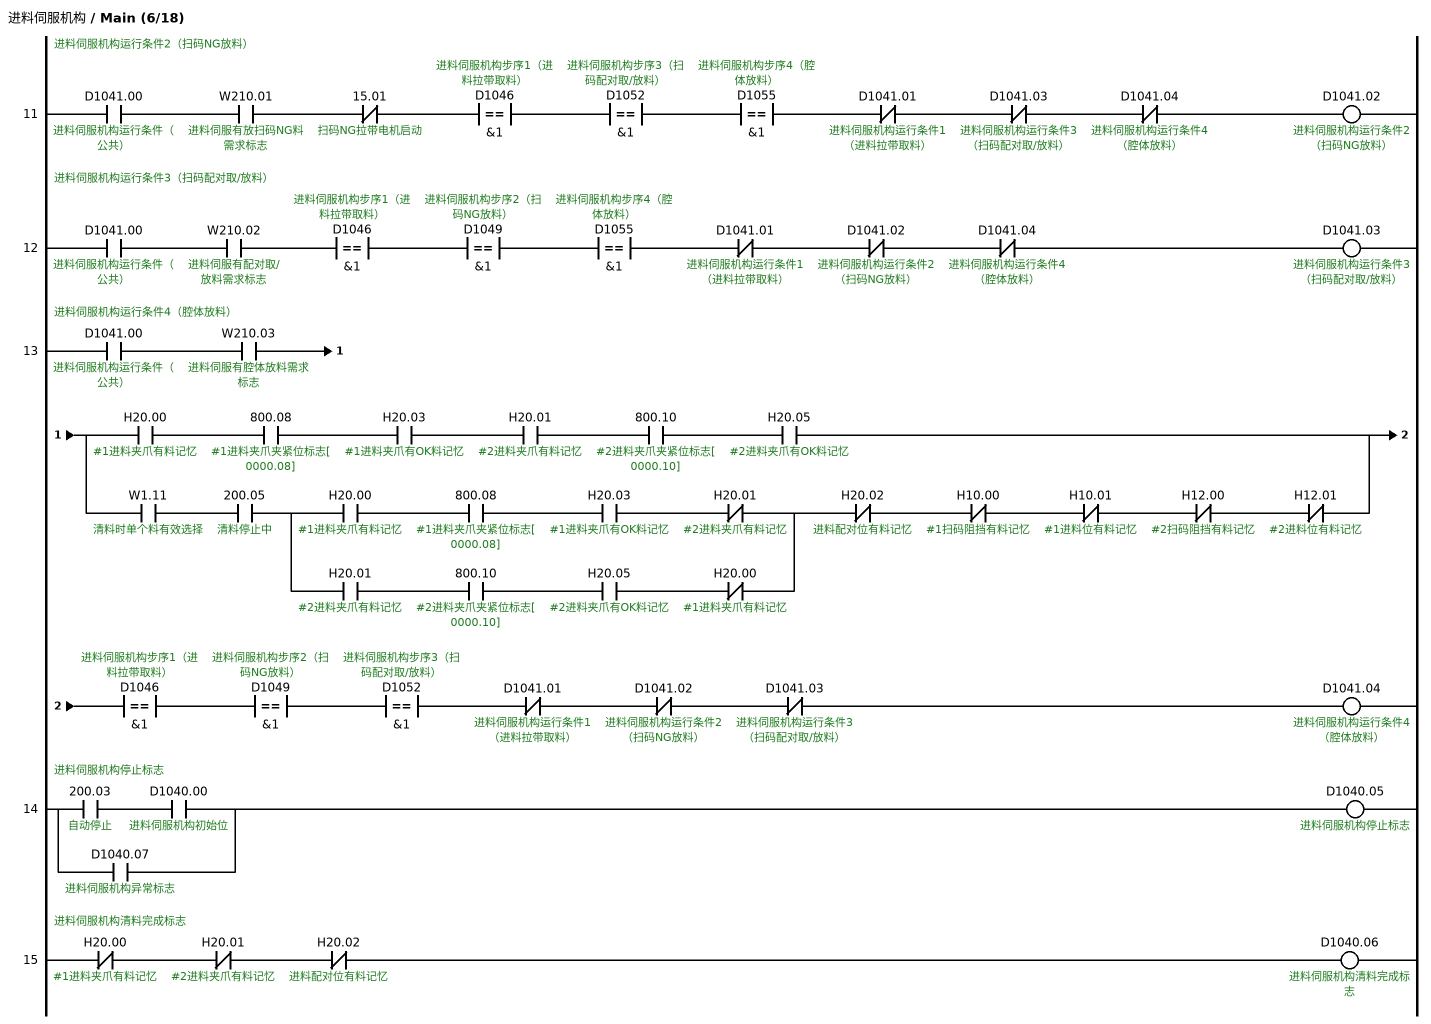
; rung 11: 进料伺服机构运行条件2（扫码NG放料）
LD D1041.00  ; 进料伺服机构运行条件（公共）
AND W210.01  ; 进料伺服有放扫码NG料需求标志
ANDNOT 15.01  ; 扫码NG拉带电机启动
AND=(300) D1046 &1  ; 进料伺服机构步序1（进料拉带取料）
AND=(300) D1052 &1  ; 进料伺服机构步序3（扫码配对取/放料）
AND=(300) D1055 &1  ; 进料伺服机构步序4（腔体放料）
ANDNOT D1041.01  ; 进料伺服机构运行条件1（进料拉带取料）
ANDNOT D1041.03  ; 进料伺服机构运行条件3（扫码配对取/放料）
ANDNOT D1041.04  ; 进料伺服机构运行条件4（腔体放料）
OUT D1041.02  ; 进料伺服机构运行条件2（扫码NG放料）
; rung 12: 进料伺服机构运行条件3（扫码配对取/放料）
LD D1041.00  ; 进料伺服机构运行条件（公共）
AND W210.02  ; 进料伺服有配对取/放料需求标志
AND=(300) D1046 &1  ; 进料伺服机构步序1（进料拉带取料）
AND=(300) D1049 &1  ; 进料伺服机构步序2（扫码NG放料）
AND=(300) D1055 &1  ; 进料伺服机构步序4（腔体放料）
ANDNOT D1041.01  ; 进料伺服机构运行条件1（进料拉带取料）
ANDNOT D1041.02  ; 进料伺服机构运行条件2（扫码NG放料）
ANDNOT D1041.04  ; 进料伺服机构运行条件4（腔体放料）
OUT D1041.03  ; 进料伺服机构运行条件3（扫码配对取/放料）
; rung 13: 进料伺服机构运行条件4（腔体放料）
LD D1041.00  ; 进料伺服机构运行条件（公共）
AND W210.03  ; 进料伺服有腔体放料需求标志
LD H20.00  ; #1进料夹爪有料记忆
AND 800.08  ; #1进料夹爪夹紧位标志[0000.08]
AND H20.03  ; #1进料夹爪有OK料记忆
AND H20.01  ; #2进料夹爪有料记忆
AND 800.10  ; #2进料夹爪夹紧位标志[0000.10]
AND H20.05  ; #2进料夹爪有OK料记忆
LD W1.11  ; 清料时单个料有效选择
AND 200.05  ; 清料停止中
LD H20.00  ; #1进料夹爪有料记忆
AND 800.08  ; #1进料夹爪夹紧位标志[0000.08]
AND H20.03  ; #1进料夹爪有OK料记忆
ANDNOT H20.01  ; #2进料夹爪有料记忆
LD H20.01  ; #2进料夹爪有料记忆
AND 800.10  ; #2进料夹爪夹紧位标志[0000.10]
AND H20.05  ; #2进料夹爪有OK料记忆
ANDNOT H20.00  ; #1进料夹爪有料记忆
ORLD
ANDLD
ANDNOT H20.02  ; 进料配对位有料记忆
ANDNOT H10.00  ; #1扫码阻挡有料记忆
ANDNOT H10.01  ; #1进料位有料记忆
ANDNOT H12.00  ; #2扫码阻挡有料记忆
ANDNOT H12.01  ; #2进料位有料记忆
ORLD
ANDLD
AND=(300) D1046 &1  ; 进料伺服机构步序1（进料拉带取料）
AND=(300) D1049 &1  ; 进料伺服机构步序2（扫码NG放料）
AND=(300) D1052 &1  ; 进料伺服机构步序3（扫码配对取/放料）
ANDNOT D1041.01  ; 进料伺服机构运行条件1（进料拉带取料）
ANDNOT D1041.02  ; 进料伺服机构运行条件2（扫码NG放料）
ANDNOT D1041.03  ; 进料伺服机构运行条件3（扫码配对取/放料）
OUT D1041.04  ; 进料伺服机构运行条件4（腔体放料）
; rung 14: 进料伺服机构停止标志
LD 200.03  ; 自动停止
AND D1040.00  ; 进料伺服机构初始位
OR D1040.07  ; 进料伺服机构异常标志
OUT D1040.05  ; 进料伺服机构停止标志
; rung 15: 进料伺服机构清料完成标志
LDNOT H20.00  ; #1进料夹爪有料记忆
ANDNOT H20.01  ; #2进料夹爪有料记忆
ANDNOT H20.02  ; 进料配对位有料记忆
OUT D1040.06  ; 进料伺服机构清料完成标志

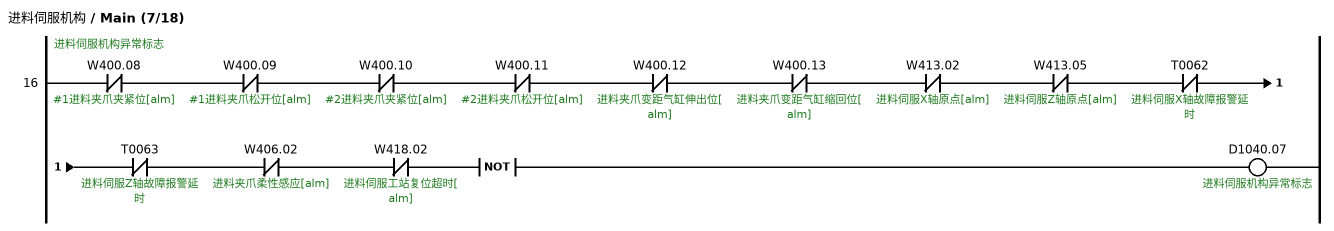
; rung 16: 进料伺服机构异常标志
LDNOT W400.08  ; #1进料夹爪夹紧位[alm]
ANDNOT W400.09  ; #1进料夹爪松开位[alm]
ANDNOT W400.10  ; #2进料夹爪夹紧位[alm]
ANDNOT W400.11  ; #2进料夹爪松开位[alm]
ANDNOT W400.12  ; 进料夹爪变距气缸伸出位[alm]
ANDNOT W400.13  ; 进料夹爪变距气缸缩回位[alm]
ANDNOT W413.02  ; 进料伺服X轴原点[alm]
ANDNOT W413.05  ; 进料伺服Z轴原点[alm]
ANDNOT T0062  ; 进料伺服X轴故障报警延时
ANDNOT T0063  ; 进料伺服Z轴故障报警延时
ANDNOT W406.02  ; 进料夹爪柔性感应[alm]
ANDNOT W418.02  ; 进料伺服工站复位超时[alm]
NOT(520)
OUT D1040.07  ; 进料伺服机构异常标志

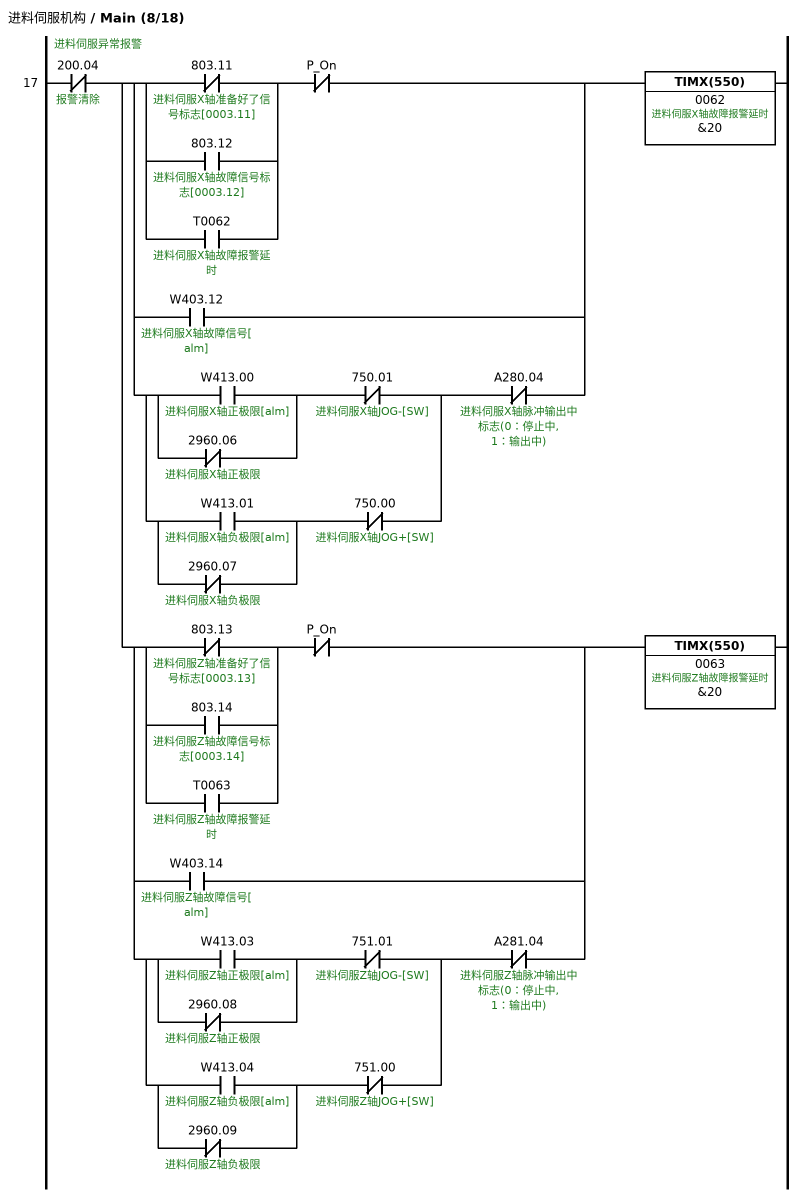
; rung 17: 进料伺服异常报警
LDNOT 200.04  ; 报警清除
OUT TR0
LDNOT 803.11  ; 进料伺服X轴准备好了信号标志[0003.11]
OR 803.12  ; 进料伺服X轴故障信号标志[0003.12]
OR T0062  ; 进料伺服X轴故障报警延时
ANDNOT P_On
OR W403.12  ; 进料伺服X轴故障信号[alm]
LD W413.00  ; 进料伺服X轴正极限[alm]
ORNOT 2960.06  ; 进料伺服X轴正极限
ANDNOT 750.01  ; 进料伺服X轴JOG-[SW]
LD W413.01  ; 进料伺服X轴负极限[alm]
ORNOT 2960.07  ; 进料伺服X轴负极限
ANDNOT 750.00  ; 进料伺服X轴JOG+[SW]
ORLD
ANDNOT A280.04  ; 进料伺服X轴脉冲输出中标志(0：停止中,1：输出中)
ORLD
ANDLD
TIMX(550) 0062 &20  ; 进料伺服X轴故障报警延时
LD TR0
LDNOT 803.13  ; 进料伺服Z轴准备好了信号标志[0003.13]
OR 803.14  ; 进料伺服Z轴故障信号标志[0003.14]
OR T0063  ; 进料伺服Z轴故障报警延时
ANDNOT P_On
OR W403.14  ; 进料伺服Z轴故障信号[alm]
LD W413.03  ; 进料伺服Z轴正极限[alm]
ORNOT 2960.08  ; 进料伺服Z轴正极限
ANDNOT 751.01  ; 进料伺服Z轴JOG-[SW]
LD W413.04  ; 进料伺服Z轴负极限[alm]
ORNOT 2960.09  ; 进料伺服Z轴负极限
ANDNOT 751.00  ; 进料伺服Z轴JOG+[SW]
ORLD
ANDNOT A281.04  ; 进料伺服Z轴脉冲输出中标志(0：停止中,1：输出中)
ORLD
ANDLD
TIMX(550) 0063 &20  ; 进料伺服Z轴故障报警延时

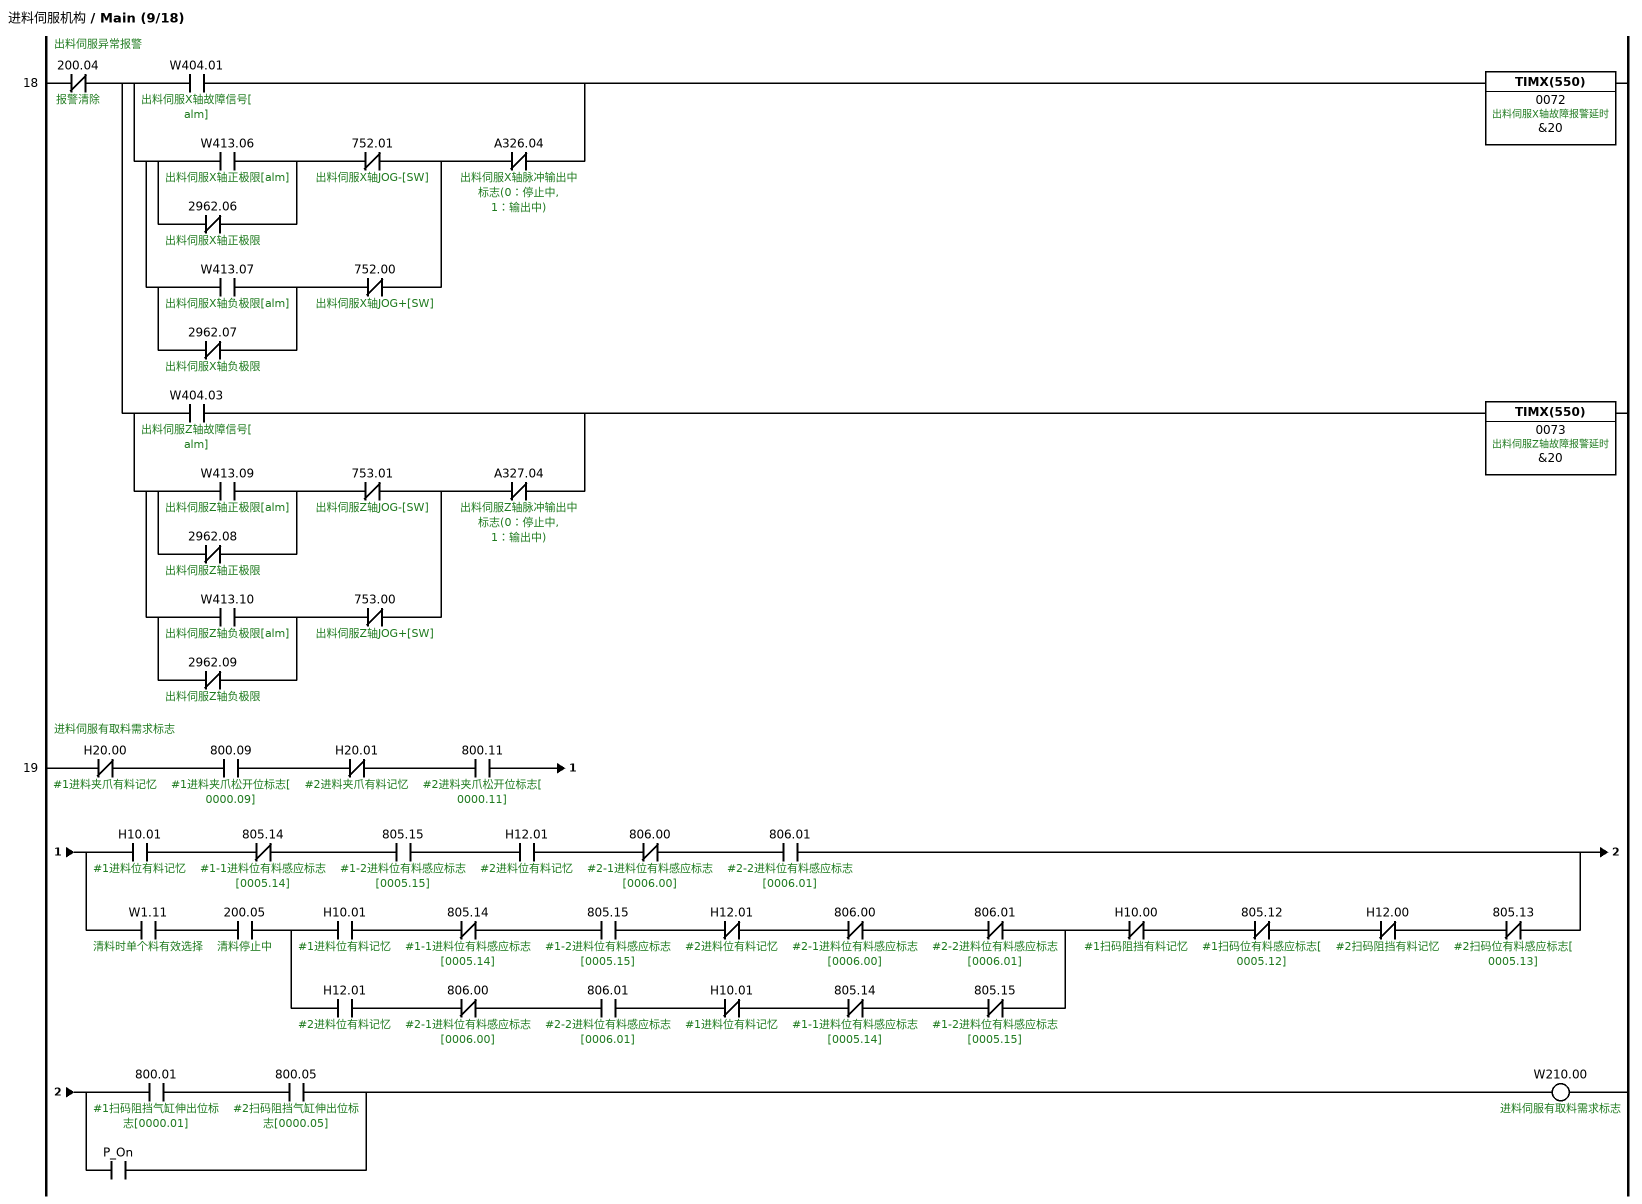
; rung 18: 出料伺服异常报警
LDNOT 200.04  ; 报警清除
OUT TR0
LD W404.01  ; 出料伺服X轴故障信号[alm]
LD W413.06  ; 出料伺服X轴正极限[alm]
ORNOT 2962.06  ; 出料伺服X轴正极限
ANDNOT 752.01  ; 出料伺服X轴JOG-[SW]
LD W413.07  ; 出料伺服X轴负极限[alm]
ORNOT 2962.07  ; 出料伺服X轴负极限
ANDNOT 752.00  ; 出料伺服X轴JOG+[SW]
ORLD
ANDNOT A326.04  ; 出料伺服X轴脉冲输出中标志(0：停止中,1：输出中)
ORLD
ANDLD
TIMX(550) 0072 &20  ; 出料伺服X轴故障报警延时
LD TR0
LD W404.03  ; 出料伺服Z轴故障信号[alm]
LD W413.09  ; 出料伺服Z轴正极限[alm]
ORNOT 2962.08  ; 出料伺服Z轴正极限
ANDNOT 753.01  ; 出料伺服Z轴JOG-[SW]
LD W413.10  ; 出料伺服Z轴负极限[alm]
ORNOT 2962.09  ; 出料伺服Z轴负极限
ANDNOT 753.00  ; 出料伺服Z轴JOG+[SW]
ORLD
ANDNOT A327.04  ; 出料伺服Z轴脉冲输出中标志(0：停止中,1：输出中)
ORLD
ANDLD
TIMX(550) 0073 &20  ; 出料伺服Z轴故障报警延时
; rung 19: 进料伺服有取料需求标志
LDNOT H20.00  ; #1进料夹爪有料记忆
AND 800.09  ; #1进料夹爪松开位标志[0000.09]
ANDNOT H20.01  ; #2进料夹爪有料记忆
AND 800.11  ; #2进料夹爪松开位标志[0000.11]
LD H10.01  ; #1进料位有料记忆
ANDNOT 805.14  ; #1-1进料位有料感应标志[0005.14]
AND 805.15  ; #1-2进料位有料感应标志[0005.15]
AND H12.01  ; #2进料位有料记忆
ANDNOT 806.00  ; #2-1进料位有料感应标志[0006.00]
AND 806.01  ; #2-2进料位有料感应标志[0006.01]
LD W1.11  ; 清料时单个料有效选择
AND 200.05  ; 清料停止中
LD H10.01  ; #1进料位有料记忆
ANDNOT 805.14  ; #1-1进料位有料感应标志[0005.14]
AND 805.15  ; #1-2进料位有料感应标志[0005.15]
ANDNOT H12.01  ; #2进料位有料记忆
ANDNOT 806.00  ; #2-1进料位有料感应标志[0006.00]
ANDNOT 806.01  ; #2-2进料位有料感应标志[0006.01]
LD H12.01  ; #2进料位有料记忆
ANDNOT 806.00  ; #2-1进料位有料感应标志[0006.00]
AND 806.01  ; #2-2进料位有料感应标志[0006.01]
ANDNOT H10.01  ; #1进料位有料记忆
ANDNOT 805.14  ; #1-1进料位有料感应标志[0005.14]
ANDNOT 805.15  ; #1-2进料位有料感应标志[0005.15]
ORLD
ANDLD
ANDNOT H10.00  ; #1扫码阻挡有料记忆
ANDNOT 805.12  ; #1扫码位有料感应标志[0005.12]
ANDNOT H12.00  ; #2扫码阻挡有料记忆
ANDNOT 805.13  ; #2扫码位有料感应标志[0005.13]
ORLD
ANDLD
LD 800.01  ; #1扫码阻挡气缸伸出位标志[0000.01]
AND 800.05  ; #2扫码阻挡气缸伸出位标志[0000.05]
OR P_On
ANDLD
OUT W210.00  ; 进料伺服有取料需求标志

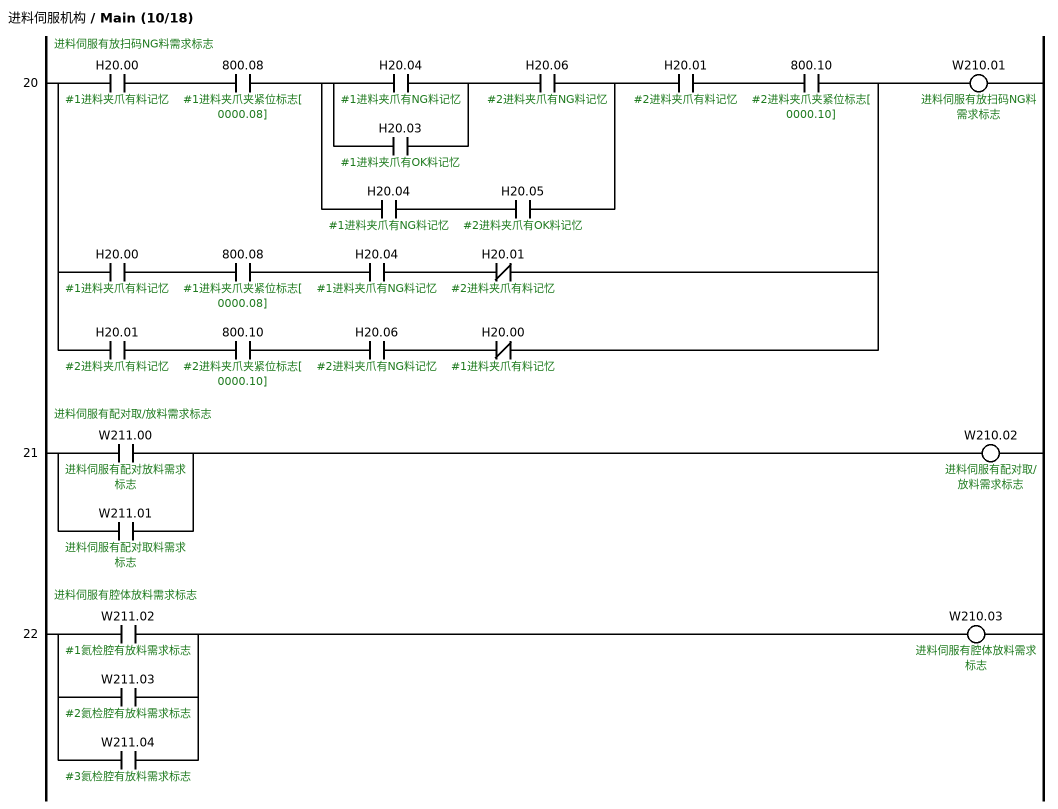
; rung 20: 进料伺服有放扫码NG料需求标志
LD H20.00  ; #1进料夹爪有料记忆
AND 800.08  ; #1进料夹爪夹紧位标志[0000.08]
LD H20.04  ; #1进料夹爪有NG料记忆
OR H20.03  ; #1进料夹爪有OK料记忆
AND H20.06  ; #2进料夹爪有NG料记忆
LD H20.04  ; #1进料夹爪有NG料记忆
AND H20.05  ; #2进料夹爪有OK料记忆
ORLD
ANDLD
AND H20.01  ; #2进料夹爪有料记忆
AND 800.10  ; #2进料夹爪夹紧位标志[0000.10]
LD H20.00  ; #1进料夹爪有料记忆
AND 800.08  ; #1进料夹爪夹紧位标志[0000.08]
AND H20.04  ; #1进料夹爪有NG料记忆
ANDNOT H20.01  ; #2进料夹爪有料记忆
ORLD
LD H20.01  ; #2进料夹爪有料记忆
AND 800.10  ; #2进料夹爪夹紧位标志[0000.10]
AND H20.06  ; #2进料夹爪有NG料记忆
ANDNOT H20.00  ; #1进料夹爪有料记忆
ORLD
OUT W210.01  ; 进料伺服有放扫码NG料需求标志
; rung 21: 进料伺服有配对取/放料需求标志
LD W211.00  ; 进料伺服有配对放料需求标志
OR W211.01  ; 进料伺服有配对取料需求标志
OUT W210.02  ; 进料伺服有配对取/放料需求标志
; rung 22: 进料伺服有腔体放料需求标志
LD W211.02  ; #1氦检腔有放料需求标志
OR W211.03  ; #2氦检腔有放料需求标志
OR W211.04  ; #3氦检腔有放料需求标志
OUT W210.03  ; 进料伺服有腔体放料需求标志

